C09060=1109.197,421.737,-96.001,-178.441,16.180,151.104
C09061=1109.203,421.984,-96.041,-178.440,16.187,151.106
C09062=1109.209,422.230,-96.081,-178.439,16.194,151.107
C09063=1109.215,422.477,-96.120,-178.437,16.202,151.109
C09064=1109.220,422.724,-96.160,-178.435,16.209,151.110
C09065=1109.225,422.971,-96.199,-178.434,16.216,151.112
C09066=1109.231,423.218,-96.238,-178.433,16.223,151.113
C09067=1109.237,423.436,-96.273,-178.432,16.230,151.115
C09068=1109.241,423.654,-96.308,-178.430,16.237,151.116
C09069=1109.246,423.872,-96.343,-178.429,16.244,151.118
C09070=1109.251,424.090,-96.378,-178.428,16.250,151.119
C09071=1109.256,424.309,-96.413,-178.426,16.257,151.120
C09072=1109.261,424.526,-96.448,-178.425,16.264,151.122
C09073=1109.266,424.744,-96.483,-178.424,16.270,151.123
C09074=1109.271,424.962,-96.518,-178.422,16.277,151.125
C09075=1109.276,425.209,-96.558,-178.421,16.285,151.127
C09076=1109.282,425.456,-96.597,-178.420,16.292,151.128
C09077=1109.287,425.703,-96.637,-178.419,16.300,151.130
C09078=1109.293,425.949,-96.677,-178.418,16.308,151.132
C09079=1109.299,426.196,-96.716,-178.416,16.316,151.133
C09080=1109.304,426.443,-96.756,-178.415,16.323,151.135
C09081=1109.310,426.689,-96.796,-178.413,16.331,151.137
C09082=1109.315,426.936,-96.836,-178.412,16.339,151.139
C09083=1109.320,427.183,-96.875,-178.411,16.347,151.140
C09084=1109.327,427.429,-96.915,-178.409,16.355,151.142
C09085=1109.332,427.676,-96.955,-178.408,16.363,151.144
C09086=1109.338,427.923,-96.995,-178.407,16.371,151.146
C09087=1109.343,428.169,-97.035,-178.406,16.379,151.147
C09088=1109.349,428.416,-97.075,-178.404,16.387,151.149
C09089=1109.354,428.663,-97.115,-178.403,16.395,151.151
C09090=1109.360,428.909,-97.155,-178.402,16.403,151.153
C09091=1109.366,429.157,-97.195,-178.401,16.411,151.155
C09092=1109.371,429.402,-97.235,-178.400,16.419,151.156
C09093=1109.377,429.650,-97.275,-178.398,16.427,151.158
C09094=1109.383,429.896,-97.315,-178.397,16.436,151.160
C09095=1109.388,430.142,-97.355,-178.396,16.444,151.162
C09096=1109.394,430.390,-97.395,-178.395,16.452,151.164
C09097=1109.399,430.636,-97.435,-178.394,16.460,151.166
C09098=1109.405,430.883,-97.475,-178.393,16.469,151.168
C09099=1109.410,431.129,-97.515,-178.392,16.477,151.170
C09100=1109.416,431.376,-97.555,-178.391,16.485,151.172
C09101=1109.422,431.623,-97.596,-178.389,16.495,151.174
C09102=1109.427,431.869,-97.635,-178.388,16.503,151.176
C09103=1109.433,432.116,-97.676,-178.387,16.511,151.178
C09104=1109.438,432.362,-97.716,-178.387,16.520,151.180
C09105=1109.444,432.609,-97.756,-178.386,16.528,151.182
C09106=1109.449,432.856,-97.797,-178.385,16.537,151.184
C09107=1109.455,433.102,-97.837,-178.384,16.545,151.186
C09108=1109.461,433.349,-97.877,-178.383,16.554,151.188
C09109=1109.467,433.595,-97.918,-178.381,16.563,151.190
C09110=1109.472,433.842,-97.958,-178.381,16.572,151.192
C09111=1109.477,434.089,-97.998,-178.380,16.580,151.194
C09112=1109.483,434.335,-98.038,-178.379,16.589,151.196
C09113=1109.488,434.582,-98.079,-178.378,16.597,151.198
C09114=1109.494,434.828,-98.119,-178.377,16.607,151.200
C09115=1109.499,435.075,-98.160,-178.376,16.616,151.202
C09116=1109.505,435.321,-98.201,-178.375,16.624,151.204
C09117=1109.510,435.568,-98.241,-178.375,16.633,151.206
C09118=1109.516,435.814,-98.281,-178.374,16.643,151.208
C09119=1109.522,436.061,-98.322,-178.373,16.652,151.211
C09120=1109.527,436.307,-98.362,-178.372,16.661,151.213
C09121=1109.532,436.554,-98.403,-178.371,16.670,151.215
C09122=1109.538,436.801,-98.444,-178.370,16.679,151.217
C09123=1109.544,437.031,-98.481,-178.369,16.688,151.219
C09124=1109.548,437.262,-98.519,-178.369,16.696,151.221
C09125=1109.553,437.492,-98.558,-178.369,16.704,151.223
C09126=1109.559,437.722,-98.596,-178.368,16.713,151.225
C09127=1109.564,437.953,-98.634,-178.367,16.722,151.227
C09128=1109.570,438.184,-98.672,-178.366,16.731,151.230
C09129=1109.574,438.414,-98.710,-178.366,16.739,151.232
C09130=1109.580,438.646,-98.748,-178.365,16.748,151.234
C09131=1109.585,438.892,-98.789,-178.365,16.758,151.236
C09132=1109.591,439.138,-98.830,-178.363,16.767,151.238
C09133=1109.597,439.385,-98.870,-178.363,16.776,151.241
C09134=1109.602,439.631,-98.911,-178.362,16.786,151.243
C09135=1109.608,439.878,-98.952,-178.362,16.796,151.246
C09136=1109.614,440.124,-98.993,-178.362,16.805,151.248
C09137=1109.619,440.371,-99.034,-178.360,16.815,151.250
C09138=1109.625,440.617,-99.074,-178.360,16.824,151.252
C09139=1109.630,440.863,-99.116,-178.359,16.835,151.255
C09140=1109.636,441.110,-99.156,-178.359,16.844,151.257
C09141=1109.641,441.357,-99.198,-178.359,16.853,151.260
C09142=1109.647,441.603,-99.239,-178.358,16.864,151.262
C09143=1109.652,441.849,-99.279,-178.358,16.873,151.265
C09144=1109.658,442.096,-99.320,-178.357,16.884,151.267
C09145=1109.664,442.342,-99.362,-178.357,16.893,151.270
C09146=1109.669,442.589,-99.402,-178.356,16.904,151.272
C09147=1109.675,442.835,-99.443,-178.356,16.913,151.275
C09148=1109.680,443.081,-99.484,-178.355,16.924,151.277
C09149=1109.685,443.328,-99.526,-178.355,16.933,151.280
C09150=1109.691,443.575,-99.567,-178.355,16.944,151.282
C09151=1109.696,443.820,-99.608,-178.355,16.954,151.285
C09152=1109.702,444.067,-99.649,-178.355,16.964,151.287
C09153=1109.707,444.314,-99.691,-178.355,16.974,151.290
C09154=1109.713,444.560,-99.732,-178.355,16.984,151.293
C09155=1109.719,444.807,-99.773,-178.356,16.994,151.295
C09156=1109.725,445.053,-99.815,-178.356,17.004,151.298
C09157=1109.729,445.299,-99.856,-178.356,17.014,151.301
C09158=1109.735,445.545,-99.897,-178.357,17.024,151.303
C09159=1109.741,445.792,-99.938,-178.358,17.034,151.306
C09160=1109.747,446.038,-99.979,-178.359,17.044,151.309
C09161=1109.752,446.285,-100.021,-178.360,17.053,151.311
C09162=1109.757,446.532,-100.062,-178.361,17.064,151.314
C09163=1109.763,446.778,-100.104,-178.362,17.074,151.317
C09164=1109.768,447.024,-100.145,-178.363,17.084,151.320
C09165=1109.774,447.270,-100.187,-178.364,17.093,151.323
C09166=1109.779,447.517,-100.228,-178.366,17.103,151.326
C09167=1109.785,447.763,-100.269,-178.367,17.113,151.328
C09168=1109.790,448.010,-100.311,-178.369,17.123,151.331
C09169=1109.796,448.257,-100.352,-178.371,17.133,151.334
C09170=1109.802,448.503,-100.394,-178.372,17.143,151.337
C09171=1109.807,448.749,-100.436,-178.375,17.152,151.340
C09172=1109.813,448.996,-100.477,-178.377,17.162,151.343
C09173=1109.817,449.242,-100.518,-178.378,17.172,151.346
C09174=1109.823,449.488,-100.560,-178.381,17.182,151.349
C09175=1109.828,449.735,-100.602,-178.383,17.191,151.352
C09176=1109.834,449.981,-100.643,-178.384,17.201,151.355
C09177=1109.839,450.228,-100.684,-178.387,17.211,151.358
C09178=1109.845,450.474,-100.726,-178.389,17.221,151.361
C09179=1109.435,450.467,-100.832,-178.476,17.454,151.438
C09180=1109.430,450.221,-100.790,-178.473,17.444,151.435
C09181=1109.424,449.975,-100.749,-178.471,17.435,151.432
C09182=1109.419,449.729,-100.707,-178.469,17.424,151.429
C09183=1109.413,449.483,-100.665,-178.467,17.414,151.426
C09184=1109.408,449.235,-100.624,-178.465,17.405,151.423
C09185=1109.402,448.989,-100.582,-178.463,17.395,151.420
C09186=1109.397,448.743,-100.540,-178.461,17.385,151.417
C09187=1109.391,448.496,-100.499,-178.459,17.375,151.414
C09188=1109.386,448.250,-100.457,-178.458,17.365,151.411
C09189=1109.380,448.003,-100.416,-178.456,17.355,151.409
C09190=1109.374,447.757,-100.375,-178.454,17.345,151.406
C09191=1109.369,447.510,-100.333,-178.453,17.335,151.403
C09192=1109.363,447.264,-100.291,-178.451,17.325,151.400
C09193=1109.358,447.017,-100.250,-178.450,17.316,151.397
C09194=1109.353,446.772,-100.209,-178.449,17.306,151.394
C09195=1109.348,446.525,-100.167,-178.448,17.295,151.391
C09196=1109.342,446.279,-100.125,-178.447,17.285,151.389
C09197=1109.336,446.032,-100.084,-178.446,17.275,151.386
C09198=1109.331,445.785,-100.042,-178.445,17.265,151.383
C09199=1109.325,445.539,-100.001,-178.444,17.255,151.380
C09200=1109.319,445.292,-99.960,-178.443,17.245,151.378
C09201=1109.314,445.046,-99.918,-178.443,17.235,151.375
C09202=1109.308,444.800,-99.877,-178.443,17.225,151.372
C09203=1109.303,444.554,-99.836,-178.443,17.215,151.370
C09204=1109.297,444.307,-99.795,-178.443,17.205,151.367
C09205=1109.292,444.061,-99.753,-178.442,17.195,151.364
C09206=1109.286,443.814,-99.712,-178.442,17.184,151.362
C09207=1109.280,443.568,-99.671,-178.442,17.174,151.359
C09208=1109.275,443.321,-99.630,-178.443,17.164,151.357
C09209=1109.270,443.075,-99.588,-178.443,17.154,151.354
C09210=1109.264,442.828,-99.547,-178.444,17.143,151.352
C09211=1109.258,442.582,-99.506,-178.444,17.134,151.349
C09212=1109.253,442.336,-99.464,-178.445,17.124,151.347
C09213=1109.247,442.089,-99.424,-178.445,17.114,151.344
C09214=1109.242,441.844,-99.383,-178.446,17.103,151.342
C09215=1109.236,441.597,-99.342,-178.446,17.094,151.339
C09216=1109.231,441.350,-99.301,-178.447,17.083,151.337
C09217=1109.225,441.104,-99.259,-178.447,17.074,151.334
C09218=1109.220,440.857,-99.219,-178.448,17.064,151.332
C09219=1109.214,440.611,-99.177,-178.448,17.054,151.329
C09220=1109.208,440.364,-99.137,-178.449,17.044,151.327
C09221=1109.203,440.118,-99.096,-178.449,17.034,151.325
C09222=1109.197,439.871,-99.054,-178.451,17.025,151.322
C09223=1109.192,439.625,-99.014,-178.451,17.015,151.320
C09224=1109.186,439.378,-98.973,-178.451,17.006,151.318
C09225=1109.180,439.132,-98.932,-178.452,16.996,151.315
C09226=1109.175,438.885,-98.891,-178.453,16.987,151.313
C09227=1109.169,438.639,-98.851,-178.454,16.977,151.311
C09228=1109.164,438.410,-98.812,-178.454,16.968,151.309
C09229=1109.159,438.181,-98.774,-178.455,16.960,151.306
C09230=1109.153,437.952,-98.737,-178.455,16.951,151.304
C09231=1109.148,437.721,-98.699,-178.456,16.942,151.302
C09232=1109.143,437.492,-98.661,-178.457,16.933,151.300
C09233=1109.138,437.263,-98.623,-178.458,16.924,151.298
C09234=1109.133,437.034,-98.585,-178.458,16.916,151.296
C09235=1109.128,436.805,-98.547,-178.459,16.907,151.294
C09236=1109.122,436.558,-98.506,-178.460,16.898,151.292
C09237=1109.116,436.311,-98.465,-178.461,16.889,151.289
C09238=1109.110,436.065,-98.425,-178.462,16.879,151.287
C09239=1109.105,435.819,-98.385,-178.463,16.871,151.285
C09240=1109.099,435.572,-98.344,-178.463,16.862,151.283
C09241=1109.094,435.325,-98.303,-178.465,16.852,151.281
C09242=1109.089,435.079,-98.263,-178.466,16.843,151.279
C09243=1109.083,434.832,-98.222,-178.466,16.834,151.277
C09244=1109.077,434.585,-98.182,-178.467,16.825,151.274
C09245=1109.072,434.339,-98.141,-178.468,16.816,151.272
C09246=1109.066,434.092,-98.101,-178.469,16.807,151.270
C09247=1109.061,433.846,-98.061,-178.470,16.799,151.268
C09248=1109.056,433.599,-98.021,-178.471,16.790,151.266
C09249=1109.050,433.352,-97.980,-178.472,16.780,151.264
C09250=1109.044,433.106,-97.940,-178.473,16.772,151.262
C09251=1109.039,432.859,-97.899,-178.474,16.763,151.260
C09252=1109.033,432.613,-97.859,-178.475,16.755,151.258
C09253=1109.028,432.367,-97.818,-178.476,16.746,151.256
C09254=1109.022,432.120,-97.778,-178.477,16.738,151.254
C09255=1109.016,431.873,-97.738,-178.479,16.729,151.252
C09256=1109.011,431.626,-97.698,-178.480,16.720,151.250
C09257=1109.005,431.380,-97.658,-178.481,16.712,151.248
C09258=1109.000,431.134,-97.617,-178.482,16.703,151.246
C09259=1108.994,430.887,-97.578,-178.483,16.695,151.244
C09260=1108.988,430.640,-97.537,-178.484,16.687,151.242
C09261=1108.983,430.394,-97.497,-178.485,16.678,151.240
C09262=1108.977,430.147,-97.457,-178.486,16.670,151.239
C09263=1108.972,429.900,-97.417,-178.487,16.662,151.237
C09264=1108.966,429.654,-97.376,-178.489,16.653,151.235
C09265=1108.960,429.406,-97.337,-178.490,16.645,151.233
C09266=1108.955,429.160,-97.296,-178.491,16.636,151.231
C09267=1108.949,428.913,-97.257,-178.493,16.628,151.229
C09268=1108.944,428.667,-97.216,-178.494,16.620,151.227
C09269=1108.938,428.420,-97.177,-178.495,16.612,151.225
C09270=1108.932,428.173,-97.136,-178.496,16.604,151.224
C09271=1108.926,427.927,-97.097,-178.497,16.596,151.222
C09272=1108.921,427.680,-97.057,-178.499,16.588,151.220
C09273=1108.916,427.433,-97.017,-178.500,16.580,151.218
C09274=1108.909,427.187,-96.977,-178.501,16.572,151.216
C09275=1108.905,426.940,-96.938,-178.503,16.564,151.215
C09276=1108.898,426.694,-96.897,-178.504,16.556,151.213
C09277=1108.893,426.446,-96.857,-178.505,16.548,151.211
C09278=1108.887,426.200,-96.818,-178.507,16.540,151.210
C09279=1108.882,425.953,-96.778,-178.508,16.532,151.208
C09280=1108.876,425.707,-96.739,-178.509,16.525,151.206
C09281=1108.870,425.460,-96.698,-178.510,16.517,151.204
C09282=1108.865,425.213,-96.659,-178.512,16.509,151.203
C09283=1108.859,424.966,-96.619,-178.513,16.501,151.201
C09284=1108.854,424.748,-96.584,-178.514,16.495,151.199
C09285=1108.849,424.530,-96.549,-178.516,16.487,151.198
C09286=1108.845,424.312,-96.514,-178.517,16.481,151.197
C09287=1108.840,424.094,-96.479,-178.518,16.474,151.195
C09288=1108.835,423.876,-96.444,-178.519,16.467,151.194
C09289=1108.830,423.657,-96.409,-178.521,16.460,151.192
C09290=1108.825,423.439,-96.374,-178.522,16.454,151.191
C09291=1108.820,423.222,-96.339,-178.524,16.447,151.189
C09292=1108.814,422.974,-96.299,-178.525,16.439,151.188
C09293=1108.809,422.728,-96.260,-178.527,16.432,151.186
C09294=1108.803,422.480,-96.220,-178.528,16.425,151.184
C09295=1108.798,422.234,-96.181,-178.529,16.417,151.183
C09296=1108.792,421.987,-96.142,-178.531,16.410,151.181
C09297=1108.786,421.740,-96.103,-178.533,16.403,151.180
C09298=1108.780,421.493,-96.063,-178.535,16.395,151.178
C09299=1108.775,421.247,-96.024,-178.535,16.388,151.177
C09300=1108.769,421.000,-95.983,-178.537,16.381,151.175
C09301=1108.764,420.754,-95.944,-178.539,16.373,151.174
C09302=1108.757,420.507,-95.905,-178.541,16.366,151.172
C09303=1108.752,420.260,-95.866,-178.542,16.359,151.171
C09304=1108.746,420.012,-95.827,-178.544,16.352,151.169
C09305=1108.742,419.766,-95.787,-178.545,16.345,151.168
C09306=1108.736,419.519,-95.748,-178.547,16.337,151.166
C09307=1108.730,419.272,-95.709,-178.548,16.331,151.165
C09308=1108.724,419.026,-95.670,-178.550,16.323,151.163
C09309=1108.718,418.778,-95.630,-178.552,16.316,151.162
C09310=1108.713,418.532,-95.591,-178.553,16.309,151.160
C09311=1108.707,418.286,-95.552,-178.555,16.302,151.159
C09312=1108.701,418.038,-95.513,-178.557,16.295,151.157
C09313=1108.696,417.791,-95.475,-178.558,16.289,151.156
C09314=1108.691,417.544,-95.435,-178.560,16.281,151.155
C09315=1108.685,417.298,-95.395,-178.562,16.274,151.153
C09316=1108.680,417.051,-95.356,-178.563,16.268,151.152
C09317=1108.674,416.803,-95.318,-178.565,16.261,151.150
C09318=1108.669,416.557,-95.279,-178.566,16.254,151.149
C09319=1108.663,416.310,-95.239,-178.568,16.247,151.148
C09320=1108.657,416.063,-95.200,-178.570,16.240,151.146
C09321=1108.651,415.817,-95.162,-178.572,16.234,151.145
C09322=1108.645,415.569,-95.123,-178.574,16.227,151.144
C09323=1108.640,415.323,-95.084,-178.575,16.221,151.142
C09324=1108.634,415.075,-95.045,-178.577,16.213,151.141
C09325=1108.628,414.829,-95.006,-178.578,16.207,151.139
C09326=1108.623,414.582,-94.968,-178.581,16.200,151.138
C09327=1108.617,414.335,-94.928,-178.583,16.193,151.137
C09328=1108.612,414.088,-94.889,-178.584,16.187,151.136
C09329=1108.606,413.841,-94.851,-178.586,16.180,151.134
C09330=1108.600,413.594,-94.812,-178.588,16.174,151.133
C09331=1108.595,413.347,-94.774,-178.590,16.168,151.132
C09332=1108.589,413.101,-94.735,-178.591,16.161,151.131
C09333=1108.583,412.853,-94.696,-178.593,16.155,151.129
C09334=1108.578,412.607,-94.657,-178.595,16.148,151.128
C09335=1108.572,412.360,-94.619,-178.597,16.142,151.127
C09336=1108.566,412.113,-94.580,-178.599,16.135,151.125
C09337=1108.561,411.866,-94.541,-178.600,16.129,151.124
C09338=1108.556,411.619,-94.503,-178.603,16.123,151.123
C09339=1108.550,411.372,-94.464,-178.604,16.117,151.122
C09340=1108.545,411.160,-94.431,-178.606,16.111,151.121
C09341=1108.540,410.948,-94.398,-178.607,16.106,151.120
C09342=1108.535,410.736,-94.364,-178.609,16.100,151.119
C09343=1108.531,410.525,-94.332,-178.611,16.095,151.118
C09344=1108.526,410.313,-94.299,-178.612,16.090,151.117
C09345=1108.521,410.101,-94.266,-178.614,16.084,151.116
C09346=1108.516,409.890,-94.233,-178.616,16.079,151.115
C09347=1108.511,409.678,-94.200,-178.617,16.074,151.114
C09348=1108.506,409.431,-94.161,-178.620,16.067,151.113
C09349=1108.501,409.184,-94.123,-178.621,16.061,151.111
C09350=1108.495,408.936,-94.084,-178.623,16.055,151.110
C09351=1108.489,408.690,-94.046,-178.625,16.049,151.109
C09352=1108.483,408.443,-94.008,-178.627,16.043,151.108
C09353=1108.478,408.196,-93.969,-178.629,16.037,151.107
C09354=1108.472,407.949,-93.931,-178.631,16.031,151.106
C09355=1108.467,407.702,-93.893,-178.633,16.025,151.105
C09356=1108.461,407.455,-93.854,-178.635,16.019,151.104
C09357=1108.455,407.208,-93.816,-178.636,16.014,151.103
C09358=1108.450,406.961,-93.778,-178.639,16.007,151.101
C09359=1108.444,406.714,-93.739,-178.641,16.001,151.100
C09360=1108.438,406.467,-93.701,-178.642,15.996,151.099
C09361=1108.433,406.220,-93.663,-178.644,15.990,151.098
C09362=1108.427,405.973,-93.625,-178.647,15.984,151.097
C09363=1108.422,405.726,-93.587,-178.649,15.978,151.096
C09364=1108.416,405.479,-93.549,-178.650,15.972,151.095
C09365=1108.411,405.232,-93.510,-178.652,15.967,151.094
C09366=1108.405,404.985,-93.472,-178.655,15.961,151.093
C09367=1108.399,404.738,-93.434,-178.657,15.955,151.092
C09368=1108.394,404.491,-93.396,-178.659,15.949,151.091
C09369=1108.388,404.244,-93.359,-178.661,15.944,151.090
C09370=1108.382,403.997,-93.320,-178.663,15.938,151.089
C09371=1108.376,403.750,-93.282,-178.665,15.933,151.088
C09372=1108.371,403.503,-93.244,-178.667,15.927,151.087
C09373=1108.365,403.256,-93.206,-178.669,15.921,151.086
C09374=1108.360,403.008,-93.168,-178.671,15.916,151.085
C09375=1108.354,402.762,-93.131,-178.673,15.910,151.084
C09376=1108.348,402.515,-93.093,-178.675,15.905,151.083
C09377=1108.343,402.268,-93.054,-178.677,15.899,151.082
C09378=1108.337,402.021,-93.017,-178.679,15.894,151.081
C09379=1108.331,401.773,-92.979,-178.681,15.888,151.080
C09380=1108.326,401.526,-92.941,-178.683,15.883,151.080
C09381=1108.320,401.279,-92.903,-178.686,15.877,151.078
C09382=1108.314,401.032,-92.865,-178.688,15.871,151.078
C09383=1108.309,400.785,-92.828,-178.690,15.866,151.077
C09384=1108.303,400.538,-92.790,-178.692,15.861,151.076
C09385=1108.297,400.291,-92.752,-178.695,15.856,151.075
C09386=1108.292,400.044,-92.714,-178.697,15.850,151.074
C09387=1108.287,399.797,-92.677,-178.699,15.845,151.073
C09388=1108.281,399.550,-92.639,-178.701,15.840,151.072
C09389=1108.275,399.303,-92.601,-178.703,15.834,151.071
C09390=1108.270,399.056,-92.564,-178.705,15.829,151.070
C09391=1108.264,398.809,-92.526,-178.707,15.824,151.070
C09392=1108.258,398.561,-92.489,-178.710,15.819,151.069
C09393=1108.252,398.315,-92.451,-178.712,15.814,151.068
C09394=1108.247,398.068,-92.413,-178.714,15.808,151.067
C09395=1108.242,397.820,-92.376,-178.716,15.803,151.066
C09396=1108.236,397.609,-92.343,-178.718,15.799,151.066
C09397=1108.232,397.396,-92.311,-178.720,15.795,151.065
C09398=1108.227,397.185,-92.279,-178.722,15.790,151.064
C09399=1108.222,396.972,-92.247,-178.724,15.786,151.063
C09400=1108.217,396.760,-92.216,-178.726,15.781,151.063
C09401=1108.212,396.548,-92.183,-178.727,15.777,151.062
C09402=1108.208,396.336,-92.151,-178.730,15.772,151.061
C09403=1108.203,396.124,-92.118,-178.732,15.768,151.061
C09404=1108.197,395.877,-92.081,-178.734,15.763,151.060
C09405=1108.191,395.630,-92.043,-178.736,15.758,151.059
C09406=1108.186,395.383,-92.006,-178.739,15.753,151.058
C09407=1108.180,395.135,-91.969,-178.741,15.748,151.058
C09408=1108.174,394.889,-91.932,-178.742,15.744,151.057
C09409=1108.169,394.641,-91.895,-178.745,15.739,151.056
C09410=1108.163,394.395,-91.857,-178.747,15.734,151.055
C09411=1108.158,394.148,-91.820,-178.750,15.729,151.055
C09412=1108.152,393.901,-91.783,-178.752,15.724,151.054
C09413=1108.146,393.654,-91.745,-178.754,15.719,151.053
C09414=1108.141,393.406,-91.708,-178.757,15.714,151.053
C09415=1108.135,393.159,-91.671,-178.759,15.709,151.052
C09416=1108.129,392.912,-91.634,-178.762,15.704,151.051
C09417=1108.123,392.665,-91.596,-178.763,15.700,151.050
C09418=1108.118,392.418,-91.559,-178.766,15.695,151.050
C09419=1108.112,392.170,-91.522,-178.768,15.691,151.049
C09420=1108.106,391.923,-91.486,-178.771,15.686,151.048
C09421=1108.101,391.677,-91.449,-178.773,15.681,151.048
C09422=1108.095,391.430,-91.412,-178.776,15.676,151.047
C09423=1108.089,391.182,-91.374,-178.778,15.672,151.046
C09424=1108.084,390.935,-91.337,-178.780,15.667,151.046
C09425=1108.078,390.688,-91.300,-178.783,15.662,151.045
C09426=1108.072,390.441,-91.264,-178.785,15.657,151.044
C09427=1108.066,390.194,-91.226,-178.788,15.653,151.044
C09428=1108.061,389.947,-91.190,-178.790,15.649,151.043
C09429=1108.055,389.700,-91.152,-178.792,15.644,151.042
C09430=1108.050,389.452,-91.115,-178.795,15.639,151.042
C09431=1108.043,389.205,-91.079,-178.797,15.635,151.041
C09432=1108.038,388.958,-91.042,-178.800,15.630,151.041
C09433=1108.033,388.711,-91.005,-178.802,15.626,151.040
C09434=1108.027,388.464,-90.969,-178.805,15.621,151.039
C09435=1108.021,388.217,-90.932,-178.807,15.617,151.039
C09436=1108.015,387.970,-90.895,-178.810,15.612,151.038
C09437=1108.010,387.722,-90.858,-178.812,15.608,151.038
C09438=1108.004,387.476,-90.822,-178.815,15.604,151.037
C09439=1107.998,387.229,-90.785,-178.817,15.599,151.037
C09440=1107.993,386.981,-90.748,-178.820,15.594,151.036
C09441=1107.986,386.734,-90.711,-178.822,15.590,151.035
C09442=1107.981,386.487,-90.674,-178.825,15.586,151.035
C09443=1107.976,386.240,-90.637,-178.827,15.581,151.034
C09444=1107.971,385.992,-90.601,-178.830,15.577,151.034
C09445=1107.965,385.746,-90.565,-178.832,15.573,151.033
C09446=1107.959,385.498,-90.528,-178.835,15.568,151.033
C09447=1107.953,385.251,-90.492,-178.838,15.564,151.032
C09448=1107.947,385.004,-90.454,-178.840,15.559,151.032
C09449=1107.943,384.757,-90.419,-178.842,15.555,151.031
C09450=1107.936,384.510,-90.382,-178.845,15.551,151.030
C09451=1107.931,384.262,-90.345,-178.848,15.546,151.030
C09452=1107.921,383.851,-90.284,-178.852,15.540,151.029
C09453=1107.912,383.439,-90.223,-178.856,15.533,151.028
C09454=1107.903,383.027,-90.162,-178.861,15.526,151.027
C09455=1107.893,382.615,-90.103,-178.865,15.519,151.027
C09456=1107.888,382.367,-90.065,-178.867,15.515,151.026
C09457=1107.882,382.121,-90.029,-178.870,15.511,151.026
C09458=1107.877,381.873,-89.993,-178.873,15.506,151.025
C09459=1107.871,381.626,-89.957,-178.875,15.502,151.025
C09460=1107.865,381.379,-89.921,-178.878,15.498,151.024
C09461=1107.859,381.131,-89.884,-178.881,15.494,151.024
C09462=1107.853,380.884,-89.848,-178.883,15.490,151.023
C09463=1107.848,380.637,-89.812,-178.886,15.486,151.023
C09464=1107.842,380.390,-89.775,-178.888,15.483,151.023
C09465=1107.836,380.142,-89.740,-178.891,15.478,151.022
C09466=1107.831,379.896,-89.703,-178.894,15.474,151.022
C09467=1107.825,379.648,-89.667,-178.896,15.470,151.021
C09468=1107.819,379.401,-89.630,-178.899,15.466,151.021
C09469=1107.814,379.154,-89.595,-178.902,15.463,151.021
C09470=1107.808,378.906,-89.559,-178.905,15.458,151.020
C09471=1107.803,378.659,-89.522,-178.907,15.455,151.020
C09472=1107.797,378.412,-89.487,-178.910,15.451,151.019
C09473=1107.791,378.165,-89.450,-178.913,15.446,151.019
C09474=1107.786,377.917,-89.414,-178.915,15.443,151.019
C09475=1107.780,377.670,-89.379,-178.918,15.439,151.018
C09476=1107.774,377.423,-89.343,-178.921,15.435,151.018
C09477=1107.769,377.175,-89.306,-178.924,15.431,151.017
C09478=1107.763,376.928,-89.271,-178.926,15.428,151.017
C09479=1107.757,376.681,-89.234,-178.929,15.423,151.017
C09480=1107.752,376.433,-89.198,-178.931,15.420,151.016
C09481=1107.746,376.186,-89.163,-178.934,15.416,151.016
C09482=1107.740,375.939,-89.127,-178.937,15.413,151.016
C09483=1107.735,375.692,-89.091,-178.940,15.408,151.015
C09484=1107.729,375.444,-89.055,-178.942,15.405,151.015
C09485=1107.724,375.197,-89.019,-178.945,15.401,151.014
C09486=1107.718,374.950,-88.983,-178.948,15.398,151.014
C09487=1107.712,374.703,-88.948,-178.951,15.393,151.014
C09488=1107.707,374.455,-88.911,-178.953,15.390,151.014
C09489=1107.701,374.208,-88.876,-178.956,15.386,151.013
C09490=1107.695,373.961,-88.840,-178.959,15.383,151.013
C09491=1107.690,373.714,-88.805,-178.962,15.379,151.013
C09492=1107.684,373.466,-88.769,-178.964,15.375,151.012
C09493=1107.679,373.219,-88.734,-178.968,15.371,151.012
C09494=1107.672,372.971,-88.698,-178.970,15.368,151.012
C09495=1107.667,372.724,-88.662,-178.973,15.364,151.011
C09496=1107.661,372.477,-88.627,-178.976,15.361,151.011
C09497=1107.656,372.229,-88.590,-178.979,15.357,151.011
C09498=1107.650,371.982,-88.555,-178.982,15.354,151.011
C09499=1107.644,371.734,-88.519,-178.984,15.350,151.010
C09500=1107.639,371.487,-88.484,-178.987,15.347,151.010
C09501=1107.633,371.239,-88.448,-178.990,15.344,151.010
C09502=1107.627,370.993,-88.413,-178.993,15.339,151.010
C09503=1107.622,370.746,-88.377,-178.996,15.336,151.009
C09504=1107.613,370.360,-88.322,-179.000,15.331,151.009
C09505=1107.604,369.975,-88.267,-179.005,15.325,151.009
C09506=1107.595,369.590,-88.211,-179.009,15.320,151.008
C09507=1107.586,369.204,-88.156,-179.014,15.314,151.008
C09508=1107.581,368.957,-88.121,-179.016,15.311,151.008
C09509=1107.575,368.710,-88.085,-179.019,15.308,151.007
C09510=1107.570,368.462,-88.050,-179.022,15.304,151.007
C09511=1107.564,368.215,-88.015,-179.025,15.301,151.007
C09512=1107.558,367.967,-87.979,-179.028,15.298,151.007
C09513=1107.553,367.720,-87.944,-179.031,15.294,151.007
C09514=1107.548,367.472,-87.909,-179.034,15.291,151.006
C09515=1107.541,367.225,-87.874,-179.037,15.287,151.006
C09516=1107.535,366.978,-87.839,-179.040,15.284,151.006
C09517=1107.529,366.730,-87.803,-179.042,15.281,151.006
C09518=1107.524,366.483,-87.768,-179.046,15.278,151.006
C09519=1107.519,366.236,-87.733,-179.048,15.274,151.005
C09520=1107.513,365.988,-87.697,-179.051,15.271,151.005
C09521=1107.508,365.741,-87.663,-179.055,15.268,151.005
C09522=1107.502,365.494,-87.627,-179.057,15.265,151.005
C09523=1107.496,365.246,-87.593,-179.060,15.262,151.005
C09524=1107.490,364.999,-87.557,-179.063,15.258,151.005
C09525=1107.484,364.751,-87.522,-179.066,15.255,151.004
C09526=1107.479,364.503,-87.487,-179.069,15.252,151.004
C09527=1107.474,364.256,-87.452,-179.072,15.248,151.004
C09528=1107.467,364.008,-87.417,-179.075,15.246,151.004
C09529=1107.462,363.761,-87.382,-179.078,15.243,151.004
C09530=1107.457,363.514,-87.347,-179.081,15.240,151.004
C09531=1107.451,363.266,-87.312,-179.084,15.236,151.004
C09532=1107.445,363.019,-87.277,-179.087,15.233,151.004
C09533=1107.439,362.772,-87.242,-179.090,15.230,151.003
C09534=1107.434,362.524,-87.207,-179.093,15.227,151.003
C09535=1107.427,362.277,-87.172,-179.096,15.224,151.003
C09536=1107.422,362.029,-87.138,-179.099,15.221,151.003
C09537=1107.417,361.781,-87.103,-179.102,15.218,151.003
C09538=1107.410,361.534,-87.068,-179.105,15.214,151.003
C09539=1107.405,361.287,-87.033,-179.108,15.211,151.003
C09540=1107.400,361.038,-86.998,-179.111,15.209,151.003
C09541=1107.393,360.792,-86.963,-179.114,15.205,151.003
C09542=1107.388,360.544,-86.929,-179.117,15.202,151.002
C09543=1107.383,360.297,-86.894,-179.120,15.199,151.002
C09544=1107.376,360.049,-86.859,-179.123,15.197,151.002
C09545=1107.371,359.802,-86.824,-179.127,15.193,151.002
C09546=1107.365,359.554,-86.790,-179.129,15.190,151.002
C09547=1107.360,359.306,-86.755,-179.132,15.188,151.002
C09548=1107.354,359.059,-86.720,-179.135,15.185,151.002
C09549=1107.348,358.812,-86.686,-179.138,15.182,151.002
C09550=1107.343,358.564,-86.651,-179.142,15.179,151.002
C09551=1107.337,358.316,-86.617,-179.145,15.176,151.002
C09552=1107.332,358.069,-86.582,-179.148,15.173,151.002
C09553=1107.326,357.822,-86.547,-179.151,15.171,151.002
C09554=1107.320,357.574,-86.512,-179.153,15.168,151.002
C09555=1107.314,357.326,-86.478,-179.157,15.164,151.002
C09556=1107.306,356.955,-86.426,-179.162,15.160,151.002
C09557=1107.297,356.586,-86.375,-179.166,15.156,151.002
C09558=1107.288,356.215,-86.324,-179.171,15.151,151.002
C09559=1107.280,355.844,-86.272,-179.175,15.147,151.002
C09560=1107.274,355.597,-86.238,-179.179,15.145,151.002
C09561=1107.269,355.349,-86.203,-179.182,15.142,151.002
C09562=1107.263,355.102,-86.169,-179.184,15.139,151.002
C09563=1107.258,354.854,-86.134,-179.187,15.137,151.002
C09564=1107.252,354.606,-86.100,-179.191,15.133,151.002
C09565=1107.246,354.359,-86.066,-179.194,15.131,151.002
C09566=1107.241,354.111,-86.031,-179.197,15.128,151.002
C09567=1107.235,353.864,-85.997,-179.200,15.125,151.002
C09568=1107.230,353.617,-85.963,-179.203,15.123,151.002
C09569=1107.224,353.369,-85.929,-179.206,15.120,151.002
C09570=1107.218,353.121,-85.895,-179.210,15.117,151.002
C09571=1107.213,352.873,-85.860,-179.213,15.114,151.002
C09572=1107.207,352.626,-85.826,-179.216,15.112,151.002
C09573=1107.201,352.379,-85.792,-179.219,15.109,151.002
C09574=1107.196,352.131,-85.757,-179.222,15.107,151.002
C09575=1107.190,351.883,-85.724,-179.225,15.104,151.002
C09576=1107.184,351.635,-85.690,-179.228,15.101,151.002
C09577=1107.178,351.388,-85.656,-179.232,15.099,151.002
C09578=1107.173,351.140,-85.621,-179.235,15.096,151.002
C09579=1107.167,350.893,-85.587,-179.238,15.093,151.002
C09580=1107.161,350.645,-85.554,-179.242,15.091,151.002
C09581=1107.156,350.398,-85.520,-179.245,15.088,151.002
C09582=1107.150,350.150,-85.485,-179.248,15.086,151.002
C09583=1107.145,349.902,-85.452,-179.251,15.083,151.002
C09584=1107.138,349.654,-85.417,-179.254,15.081,151.002
C09585=1107.133,349.407,-85.383,-179.257,15.078,151.003
C09586=1107.127,349.159,-85.350,-179.260,15.076,151.003
C09587=1107.122,348.911,-85.315,-179.263,15.073,151.003
C09588=1107.116,348.664,-85.281,-179.267,15.071,151.003
C09589=1107.110,348.416,-85.248,-179.270,15.069,151.003
C09590=1107.105,348.169,-85.214,-179.274,15.065,151.003
C09591=1107.099,347.921,-85.180,-179.277,15.063,151.003
C09592=1107.093,347.674,-85.146,-179.280,15.060,151.003
C09593=1107.088,347.426,-85.113,-179.283,15.058,151.003
C09594=1107.083,347.178,-85.078,-179.287,15.056,151.003
C09595=1107.077,346.930,-85.045,-179.290,15.053,151.004
C09596=1107.071,346.683,-85.011,-179.293,15.051,151.004
C09597=1107.066,346.435,-84.978,-179.296,15.048,151.004
C09598=1107.060,346.188,-84.943,-179.299,15.046,151.004
C09599=1107.054,345.940,-84.910,-179.302,15.043,151.004
C09600=1107.048,345.693,-84.876,-179.306,15.041,151.004
C09601=1107.043,345.445,-84.843,-179.309,15.039,151.004
C09602=1107.037,345.198,-84.809,-179.312,15.036,151.004
C09603=1107.031,344.950,-84.775,-179.315,15.034,151.004
C09604=1107.025,344.701,-84.742,-179.319,15.032,151.005
C09605=1107.019,344.454,-84.708,-179.322,15.029,151.005
C09606=1107.014,344.206,-84.674,-179.325,15.027,151.005
C09607=1107.008,343.958,-84.641,-179.328,15.025,151.005
C09608=1107.000,343.590,-84.590,-179.333,15.021,151.005
C09609=1106.991,343.222,-84.541,-179.338,15.018,151.006
C09610=1106.983,342.854,-84.491,-179.343,15.014,151.006
C09611=1106.974,342.485,-84.441,-179.348,15.011,151.006
C09612=1106.969,342.237,-84.408,-179.351,15.008,151.006
C09613=1106.963,341.989,-84.374,-179.355,15.006,151.006
C09614=1106.958,341.741,-84.341,-179.358,15.004,151.007
C09615=1106.951,341.494,-84.308,-179.361,15.002,151.007
C09616=1106.946,341.246,-84.274,-179.365,14.999,151.007
C09617=1106.941,340.999,-84.241,-179.368,14.997,151.007
C09618=1106.935,340.751,-84.208,-179.371,14.995,151.007
C09619=1106.930,340.503,-84.175,-179.375,14.993,151.007
C09620=1106.924,340.255,-84.141,-179.378,14.990,151.007
C09621=1106.918,340.008,-84.107,-179.381,14.989,151.008
C09622=1106.912,339.760,-84.075,-179.384,14.987,151.008
C09623=1106.906,339.513,-84.041,-179.387,14.984,151.008
C09624=1106.901,339.265,-84.008,-179.391,14.982,151.008
C09625=1106.895,339.017,-83.974,-179.394,14.980,151.008
C09626=1106.890,338.769,-83.941,-179.397,14.978,151.009
C09627=1106.883,338.521,-83.908,-179.401,14.976,151.009
C09628=1106.878,338.274,-83.875,-179.404,14.973,151.009
C09629=1106.873,338.026,-83.842,-179.408,14.971,151.009
C09630=1106.867,337.778,-83.809,-179.411,14.969,151.010
C09631=1106.861,337.531,-83.776,-179.415,14.967,151.010
C09632=1106.855,337.283,-83.743,-179.418,14.965,151.010
C09633=1106.850,337.035,-83.709,-179.421,14.963,151.010
C09634=1106.844,336.787,-83.677,-179.424,14.962,151.011
C09635=1106.838,336.539,-83.643,-179.427,14.959,151.011
C09636=1106.833,336.291,-83.611,-179.431,14.957,151.011
C09637=1106.827,336.044,-83.578,-179.434,14.955,151.011
C09638=1106.821,335.796,-83.545,-179.438,14.953,151.011
C09639=1106.816,335.548,-83.512,-179.441,14.951,151.012
C09640=1106.810,335.300,-83.479,-179.445,14.949,151.012
C09641=1106.804,335.053,-83.446,-179.448,14.947,151.012
C09642=1106.799,334.805,-83.412,-179.452,14.945,151.013
C09643=1106.793,334.557,-83.381,-179.454,14.943,151.013
C09644=1106.788,334.309,-83.347,-179.458,14.941,151.013
C09645=1106.781,334.062,-83.314,-179.461,14.939,151.013
C09646=1106.776,333.814,-83.281,-179.465,14.937,151.013
C09647=1106.771,333.565,-83.248,-179.468,14.935,151.014
C09648=1106.765,333.318,-83.216,-179.472,14.933,151.014
C09649=1106.759,333.070,-83.183,-179.475,14.931,151.014
C09650=1106.753,332.822,-83.151,-179.478,14.929,151.014
C09651=1106.748,332.574,-83.117,-179.481,14.927,151.015
C09652=1106.742,332.327,-83.085,-179.485,14.925,151.015
C09653=1106.737,332.079,-83.052,-179.489,14.923,151.015
C09654=1106.730,331.831,-83.020,-179.492,14.921,151.016
C09655=1106.725,331.583,-82.986,-179.496,14.919,151.016
C09656=1106.719,331.335,-82.954,-179.499,14.918,151.016
C09657=1106.713,331.088,-82.922,-179.502,14.916,151.017
C09658=1106.708,330.840,-82.889,-179.506,14.914,151.017
C09659=1106.702,330.592,-82.857,-179.509,14.912,151.017
C09660=1106.693,330.218,-82.807,-179.515,14.909,151.018
C09661=1106.684,329.843,-82.758,-179.519,14.907,151.018
C09662=1106.675,329.469,-82.709,-179.525,14.904,151.019
C09663=1106.667,329.095,-82.660,-179.530,14.901,151.019
C09664=1106.661,328.846,-82.627,-179.534,14.899,151.019
C09665=1106.655,328.598,-82.595,-179.536,14.898,151.020
C09666=1106.649,328.350,-82.562,-179.540,14.896,151.020
C09667=1106.644,328.103,-82.530,-179.544,14.894,151.021
C09668=1106.638,327.855,-82.497,-179.547,14.892,151.021
C09669=1106.632,327.607,-82.465,-179.550,14.891,151.021
C09670=1106.627,327.360,-82.432,-179.554,14.889,151.021
C09671=1106.621,327.111,-82.400,-179.557,14.887,151.022
C09672=1106.615,326.863,-82.368,-179.561,14.885,151.022
C09673=1106.609,326.616,-82.335,-179.565,14.883,151.022
C09674=1106.604,326.368,-82.303,-179.568,14.882,151.023
C09675=1106.598,326.119,-82.271,-179.571,14.880,151.023
C09676=1106.592,325.872,-82.238,-179.575,14.878,151.024
C09677=1106.587,325.624,-82.207,-179.578,14.877,151.024
C09678=1106.581,325.376,-82.174,-179.581,14.875,151.024
C09679=1106.575,325.128,-82.141,-179.585,14.874,151.025
C09680=1106.570,324.881,-82.110,-179.589,14.872,151.025
C09681=1106.564,324.633,-82.078,-179.592,14.870,151.025
C09682=1106.558,324.385,-82.046,-179.595,14.869,151.026
C09683=1106.553,324.136,-82.013,-179.599,14.867,151.026
C09684=1106.547,323.889,-81.981,-179.603,14.865,151.026
C09685=1106.541,323.641,-81.949,-179.606,14.864,151.027
C09686=1106.535,323.393,-81.917,-179.609,14.862,151.027
C09687=1106.530,323.146,-81.885,-179.613,14.860,151.028
C09688=1106.524,322.897,-81.853,-179.617,14.858,151.028
C09689=1106.519,322.649,-81.821,-179.620,14.857,151.028
C09690=1106.513,322.402,-81.788,-179.623,14.855,151.029
C09691=1106.507,322.154,-81.756,-179.627,14.853,151.029
C09692=1106.502,321.906,-81.725,-179.631,14.852,151.029
C09693=1106.496,321.658,-81.693,-179.634,14.851,151.030
C09694=1106.490,321.411,-81.661,-179.637,14.849,151.030
C09695=1106.484,321.162,-81.629,-179.641,14.847,151.031
C09696=1106.479,320.915,-81.597,-179.644,14.846,151.031
C09697=1106.474,320.666,-81.565,-179.648,14.844,151.031
C09698=1106.468,320.419,-81.533,-179.651,14.842,151.032
C09699=1106.462,320.171,-81.501,-179.654,14.841,151.032
C09700=1106.457,319.923,-81.469,-179.658,14.840,151.032
C09701=1106.451,319.675,-81.437,-179.662,14.838,151.033
C09702=1106.446,319.427,-81.406,-179.666,14.836,151.033
C09703=1106.440,319.179,-81.374,-179.669,14.835,151.034
C09704=1106.434,318.932,-81.342,-179.672,14.833,151.034
C09705=1106.428,318.683,-81.310,-179.676,14.831,151.034
C09706=1106.423,318.436,-81.278,-179.679,14.830,151.035
C09707=1106.417,318.187,-81.247,-179.683,14.828,151.035
C09708=1106.412,317.940,-81.215,-179.687,14.827,151.036
C09709=1106.406,317.691,-81.183,-179.690,14.826,151.036
C09710=1106.400,317.444,-81.152,-179.693,14.824,151.037
C09711=1106.394,317.196,-81.120,-179.697,14.822,151.037
C09712=1106.386,316.814,-81.071,-179.702,14.820,151.037
C09713=1106.377,316.433,-81.022,-179.708,14.818,151.038
C09714=1106.370,316.051,-80.973,-179.713,14.815,151.039
C09715=1106.361,315.669,-80.925,-179.718,14.813,151.039
C09716=1106.355,315.422,-80.893,-179.722,14.811,151.040
C09717=1106.349,315.173,-80.862,-179.725,14.811,151.040
C09718=1106.344,314.926,-80.831,-179.729,14.809,151.041
C09719=1106.338,314.678,-80.799,-179.733,14.808,151.041
C09720=1106.333,314.429,-80.768,-179.736,14.807,151.042
C09721=1106.326,314.181,-80.736,-179.740,14.805,151.042
C09722=1106.320,313.934,-80.705,-179.744,14.804,151.043
C09723=1106.315,313.686,-80.674,-179.747,14.802,151.043
C09724=1106.309,313.438,-80.642,-179.751,14.801,151.044
C09725=1106.303,313.190,-80.611,-179.754,14.800,151.044
C09726=1106.298,312.942,-80.579,-179.758,14.798,151.045
C09727=1106.291,312.694,-80.548,-179.762,14.797,151.045
C09728=1106.286,312.446,-80.516,-179.765,14.796,151.045
C09729=1106.280,312.198,-80.485,-179.769,14.794,151.046
C09730=1106.274,311.951,-80.454,-179.772,14.794,151.046
C09731=1106.269,311.702,-80.423,-179.776,14.792,151.047
C09732=1106.263,311.454,-80.391,-179.780,14.790,151.047
C09733=1106.257,311.207,-80.361,-179.783,14.790,151.048
C09734=1106.251,310.958,-80.329,-179.787,14.788,151.048
C09735=1106.246,310.711,-80.298,-179.790,14.787,151.049
C09736=1106.240,310.462,-80.266,-179.794,14.786,151.049
C09737=1106.235,310.214,-80.235,-179.798,14.784,151.050
C09738=1106.228,309.967,-80.204,-179.801,14.783,151.050
C09739=1106.223,309.718,-80.173,-179.805,14.782,151.051
C09740=1106.217,309.471,-80.142,-179.808,14.781,151.051
C09741=1106.212,309.223,-80.111,-179.812,14.779,151.052
C09742=1106.206,308.974,-80.080,-179.815,14.778,151.052
C09743=1106.200,308.727,-80.049,-179.819,14.777,151.053
C09744=1106.195,308.479,-80.018,-179.823,14.775,151.053
C09745=1106.189,308.231,-79.987,-179.826,14.775,151.054
C09746=1106.183,307.983,-79.955,-179.830,14.773,151.054
C09747=1106.177,307.735,-79.925,-179.833,14.772,151.055
C09748=1106.172,307.487,-79.894,-179.837,14.771,151.055
C09749=1106.166,307.240,-79.863,-179.840,14.770,151.056
C09750=1106.160,306.991,-79.832,-179.844,14.768,151.056
C09751=1106.154,306.743,-79.801,-179.848,14.767,151.057
C09752=1106.149,306.495,-79.770,-179.851,14.766,151.057
C09753=1106.143,306.248,-79.739,-179.855,14.764,151.058
C09754=1106.137,305.999,-79.708,-179.859,14.764,151.059
C09755=1106.132,305.751,-79.678,-179.863,14.762,151.059
C09756=1106.126,305.503,-79.646,-179.866,14.761,151.060
C09757=1106.120,305.256,-79.616,-179.870,14.760,151.060
C09758=1106.115,305.007,-79.585,-179.874,14.758,151.061
C09759=1106.109,304.759,-79.554,-179.877,14.757,151.061
C09760=1106.104,304.511,-79.523,-179.881,14.756,151.062
C09761=1106.098,304.263,-79.493,-179.884,14.755,151.062
C09762=1106.092,304.016,-79.462,-179.888,14.754,151.063
C09763=1106.087,303.768,-79.431,-179.891,14.753,151.063
C09764=1106.078,303.389,-79.384,-179.897,14.751,151.064
C09765=1106.070,303.009,-79.338,-179.903,14.750,151.065
C09766=1106.061,302.630,-79.290,-179.909,14.747,151.066
C09767=1106.052,302.251,-79.243,-179.914,14.746,151.066
C09768=1106.047,302.003,-79.213,-179.918,14.745,151.067
C09769=1106.041,301.755,-79.182,-179.921,14.744,151.068
C09770=1106.036,301.507,-79.151,-179.925,14.742,151.068
C09771=1106.030,301.259,-79.121,-179.928,14.741,151.069
C09772=1106.025,301.011,-79.090,-179.933,14.740,151.069
C09773=1106.019,300.763,-79.060,-179.936,14.739,151.070
C09774=1106.013,300.515,-79.029,-179.940,14.738,151.070
C09775=1106.008,300.267,-78.999,-179.943,14.737,151.071
C09776=1106.002,300.020,-78.968,-179.947,14.736,151.071
C09777=1105.997,299.771,-78.939,-179.950,14.735,151.072
C09778=1105.992,299.523,-78.908,-179.954,14.733,151.072
C09779=1105.986,299.275,-78.877,-179.957,14.733,151.073
C09780=1105.979,299.027,-78.847,-179.962,14.732,151.074
C09781=1105.974,298.779,-78.816,-179.965,14.731,151.074
C09782=1105.969,298.531,-78.785,-179.969,14.729,151.075
C09783=1105.963,298.283,-78.755,-179.972,14.729,151.075
C09784=1105.957,298.034,-78.725,-179.976,14.727,151.076
C09785=1105.951,297.787,-78.695,-179.980,14.727,151.076
C09786=1105.946,297.539,-78.665,-179.984,14.725,151.077
C09787=1105.940,297.291,-78.634,-179.987,14.724,151.077
C09788=1105.935,297.042,-78.604,-179.991,14.723,151.078
C09789=1105.929,296.794,-78.574,-179.994,14.722,151.079
C09790=1105.923,296.547,-78.543,-179.998,14.721,151.079
C09791=1105.917,296.299,-78.513,179.998,14.720,151.080
C09792=1105.912,296.050,-78.483,179.994,14.719,151.080
C09793=1105.906,295.802,-78.453,179.991,14.718,151.081
C09794=1105.900,295.555,-78.423,179.987,14.717,151.082
C09795=1105.895,295.306,-78.393,179.984,14.717,151.082
C09796=1105.889,295.058,-78.363,179.980,14.716,151.083
C09797=1105.884,294.810,-78.333,179.976,14.715,151.083
C09798=1105.878,294.562,-78.303,179.973,14.714,151.084
C09799=1105.872,294.314,-78.272,179.968,14.713,151.085
C09800=1105.866,294.066,-78.243,179.965,14.712,151.085
C09801=1105.861,293.818,-78.212,179.961,14.711,151.086
C09802=1105.855,293.570,-78.183,179.958,14.710,151.086
C09803=1105.849,293.322,-78.152,179.953,14.709,151.087
C09804=1105.844,293.073,-78.123,179.950,14.709,151.088
C09805=1105.838,292.825,-78.092,179.946,14.707,151.088
C09806=1105.832,292.577,-78.063,179.942,14.707,151.089
C09807=1105.827,292.329,-78.032,179.939,14.706,151.089
C09808=1105.821,292.081,-78.003,179.935,14.705,151.090
C09809=1105.815,291.833,-77.972,179.932,14.704,151.091
C09810=1105.810,291.585,-77.943,179.928,14.703,151.091
C09811=1105.804,291.337,-77.912,179.924,14.702,151.092
C09812=1105.798,291.088,-77.883,179.920,14.701,151.093
C09813=1105.793,290.840,-77.852,179.917,14.700,151.093
C09814=1105.787,290.592,-77.823,179.913,14.700,151.094
C09815=1105.782,290.344,-77.793,179.909,14.699,151.094
C09816=1105.773,289.979,-77.749,179.904,14.698,151.095
C09817=1105.764,289.614,-77.705,179.898,14.697,151.096
C09818=1105.756,289.249,-77.662,179.893,14.695,151.097
C09819=1105.748,288.884,-77.619,179.887,14.694,151.098
C09820=1105.742,288.636,-77.588,179.884,14.693,151.099
C09821=1105.737,288.387,-77.559,179.880,14.692,151.099
C09822=1105.731,288.139,-77.530,179.876,14.692,151.100
C09823=1105.725,287.891,-77.499,179.872,14.691,151.101
C09824=1105.719,287.643,-77.470,179.868,14.690,151.101
C09825=1105.714,287.395,-77.440,179.865,14.689,151.102
C09826=1105.708,287.146,-77.411,179.861,14.688,151.103
C09827=1105.702,286.898,-77.381,179.857,14.688,151.103
C09828=1105.697,286.651,-77.351,179.854,14.687,151.104
C09829=1105.691,286.402,-77.322,179.849,14.686,151.105
C09830=1105.685,286.154,-77.293,179.846,14.686,151.105
C09831=1105.680,285.906,-77.263,179.843,14.685,151.106
C09832=1105.674,285.657,-77.233,179.839,14.684,151.106
C09833=1105.668,285.409,-77.204,179.835,14.684,151.107
C09834=1105.662,285.161,-77.175,179.831,14.683,151.108
C09835=1105.657,284.913,-77.146,179.827,14.682,151.109
C09836=1105.652,284.665,-77.116,179.824,14.682,151.109
C09837=1105.646,284.417,-77.087,179.820,14.680,151.110
C09838=1105.640,284.169,-77.056,179.816,14.680,151.110
C09839=1105.634,283.920,-77.027,179.813,14.679,151.111
C09840=1105.629,283.673,-76.998,179.808,14.678,151.112
C09841=1105.623,283.424,-76.969,179.805,14.678,151.112
C09842=1105.617,283.176,-76.939,179.801,14.677,151.113
C09843=1105.611,282.928,-76.910,179.797,14.676,151.114
C09844=1105.606,282.679,-76.881,179.794,14.675,151.114
C09845=1105.600,282.431,-76.852,179.790,14.674,151.115
C09846=1105.595,282.183,-76.823,179.786,14.674,151.116
C09847=1105.589,281.934,-76.793,179.783,14.674,151.116
C09848=1105.583,281.686,-76.764,179.778,14.672,151.117
C09849=1105.578,281.439,-76.735,179.775,14.672,151.118
C09850=1105.572,281.190,-76.706,179.771,14.672,151.118
C09851=1105.567,280.942,-76.676,179.767,14.671,151.119
C09852=1105.560,280.694,-76.647,179.764,14.670,151.120
C09853=1105.556,280.446,-76.618,179.760,14.670,151.120
C09854=1105.549,280.197,-76.589,179.756,14.669,151.121
C09855=1105.544,279.949,-76.560,179.752,14.668,151.122
C09856=1105.538,279.701,-76.531,179.749,14.668,151.123
C09857=1105.533,279.453,-76.501,179.745,14.667,151.123
C09858=1105.527,279.204,-76.473,179.741,14.666,151.124
C09859=1105.521,278.956,-76.443,179.737,14.666,151.125
C09860=1105.515,278.708,-76.414,179.733,14.665,151.125
C09861=1105.509,278.460,-76.386,179.730,14.664,151.126
C09862=1105.504,278.211,-76.357,179.726,14.664,151.127
C09863=1105.498,277.963,-76.328,179.722,14.663,151.127
C09864=1105.493,277.715,-76.299,179.718,14.662,151.128
C09865=1105.487,277.467,-76.270,179.715,14.662,151.129
C09866=1105.482,277.218,-76.241,179.711,14.661,151.129
C09867=1105.476,276.971,-76.212,179.707,14.661,151.130
C09868=1105.467,276.615,-76.170,179.701,14.660,151.131
C09869=1105.459,276.259,-76.129,179.696,14.659,151.132
C09870=1105.452,275.903,-76.088,179.691,14.658,151.133
C09871=1105.443,275.548,-76.047,179.685,14.657,151.134
C09872=1105.438,275.299,-76.018,179.682,14.657,151.135
C09873=1105.432,275.051,-75.990,179.678,14.657,151.136
C09874=1105.426,274.803,-75.961,179.674,14.656,151.136
C09875=1105.421,274.554,-75.932,179.670,14.655,151.137
C09876=1105.415,274.307,-75.903,179.667,14.655,151.138
C09877=1105.409,274.058,-75.875,179.662,14.654,151.138
C09878=1105.404,273.809,-75.845,179.659,14.654,151.139
C09879=1105.398,273.561,-75.817,179.655,14.653,151.140
C09880=1105.392,273.313,-75.788,179.652,14.653,151.141
C09881=1105.386,273.064,-75.760,179.647,14.652,151.141
C09882=1105.381,272.817,-75.730,179.643,14.652,151.142
C09883=1105.375,272.568,-75.702,179.640,14.651,151.143
C09884=1105.370,272.321,-75.673,179.636,14.650,151.143
C09885=1105.364,272.072,-75.645,179.632,14.650,151.144
C09886=1105.358,271.823,-75.617,179.629,14.650,151.145
C09887=1105.352,271.576,-75.588,179.625,14.650,151.146
C09888=1105.347,271.327,-75.559,179.621,14.649,151.146
C09889=1105.341,271.078,-75.531,179.617,14.648,151.147
C09890=1105.335,270.830,-75.502,179.613,14.648,151.148
C09891=1105.330,270.582,-75.474,179.610,14.647,151.148
C09892=1105.324,270.334,-75.446,179.605,14.647,151.149
C09893=1105.318,270.085,-75.417,179.602,14.646,151.150
C09894=1105.313,269.837,-75.388,179.598,14.646,151.151
C09895=1105.307,269.588,-75.360,179.594,14.645,151.151
C09896=1105.302,269.340,-75.332,179.590,14.645,151.152
C09897=1105.296,269.092,-75.303,179.587,14.644,151.153
C09898=1105.290,268.844,-75.275,179.583,14.644,151.154
C09899=1105.284,268.595,-75.247,179.579,14.643,151.155
C09900=1105.279,268.347,-75.219,179.575,14.643,151.155
C09901=1105.273,268.099,-75.190,179.571,14.643,151.156
C09902=1105.267,267.850,-75.162,179.568,14.643,151.157
C09903=1105.261,267.602,-75.133,179.563,14.642,151.157
C09904=1105.255,267.354,-75.105,179.560,14.641,151.158
C09905=1105.250,267.106,-75.077,179.556,14.641,151.159
C09906=1105.244,266.857,-75.049,179.552,14.641,151.160
C09907=1105.239,266.609,-75.021,179.549,14.640,151.160
C09908=1105.233,266.360,-74.992,179.545,14.639,151.161
C09909=1105.228,266.112,-74.965,179.541,14.639,151.162
C09910=1105.222,265.864,-74.937,179.537,14.639,151.163
C09911=1105.216,265.615,-74.908,179.534,14.639,151.163
C09912=1105.211,265.367,-74.880,179.529,14.638,151.164
C09913=1105.205,265.118,-74.852,179.526,14.638,151.165
C09914=1105.200,264.870,-74.824,179.522,14.637,151.166
C09915=1105.194,264.622,-74.796,179.518,14.637,151.166
C09916=1105.188,264.373,-74.768,179.514,14.636,151.167
C09917=1105.182,264.125,-74.739,179.510,14.636,151.168
C09918=1105.176,263.877,-74.712,179.506,14.636,151.169
C09919=1105.170,263.628,-74.684,179.503,14.636,151.170
C09920=1105.162,263.276,-74.644,179.497,14.635,151.171
C09921=1105.154,262.923,-74.604,179.492,14.635,151.172
C09922=1105.146,262.570,-74.564,179.486,14.634,151.173
C09923=1105.138,262.217,-74.525,179.481,14.634,151.174
C09924=1105.132,261.968,-74.497,179.477,14.633,151.175
C09925=1105.127,261.720,-74.469,179.473,14.633,151.175
C09926=1105.120,261.472,-74.441,179.469,14.633,151.176
C09927=1105.115,261.224,-74.413,179.466,14.633,151.177
C09928=1105.110,260.975,-74.386,179.462,14.633,151.178
C09929=1105.103,260.727,-74.358,179.457,14.632,151.179
C09930=1105.098,260.479,-74.330,179.454,14.632,151.179
C09931=1105.092,260.230,-74.302,179.450,14.631,151.180
C09932=1105.086,259.982,-74.274,179.446,14.631,151.181
C09933=1105.081,259.733,-74.247,179.443,14.631,151.182
C09934=1105.075,259.485,-74.219,179.438,14.630,151.183
C09935=1105.069,259.237,-74.191,179.435,14.630,151.183
C09936=1105.063,258.988,-74.164,179.431,14.630,151.184
C09937=1105.058,258.740,-74.136,179.427,14.630,151.185
C09938=1105.052,258.491,-74.108,179.423,14.630,151.186
C09939=1105.046,258.242,-74.081,179.420,14.629,151.186
C09940=1105.041,257.994,-74.053,179.415,14.629,151.187
C09941=1105.035,257.746,-74.025,179.412,14.628,151.188
C09942=1105.029,257.497,-73.998,179.408,14.628,151.189
C09943=1105.023,257.249,-73.970,179.404,14.628,151.190
C09944=1105.018,257.001,-73.943,179.400,14.628,151.190
C09945=1105.012,256.752,-73.915,179.396,14.628,151.191
C09946=1105.006,256.504,-73.887,179.392,14.627,151.192
C09947=1105.001,256.256,-73.860,179.388,14.627,151.193
C09948=1104.995,256.007,-73.832,179.385,14.627,151.194
C09949=1104.990,255.758,-73.805,179.381,14.627,151.194
C09950=1104.984,255.511,-73.778,179.377,14.626,151.195
C09951=1104.978,255.261,-73.750,179.374,14.626,151.196
C09952=1104.972,255.013,-73.723,179.369,14.625,151.197
C09953=1104.967,254.765,-73.695,179.365,14.625,151.198
C09954=1104.961,254.517,-73.668,179.362,14.625,151.198
C09955=1104.955,254.268,-73.640,179.358,14.625,151.199
C09956=1104.950,254.020,-73.612,179.354,14.625,151.200
C09957=1104.944,253.771,-73.586,179.351,14.625,151.201
C09958=1104.939,253.523,-73.559,179.346,14.624,151.202
C09959=1104.932,253.274,-73.531,179.342,14.624,151.202
C09960=1104.927,253.025,-73.504,179.339,14.624,151.203
C09961=1104.921,252.777,-73.477,179.335,14.623,151.204
C09962=1104.916,252.529,-73.449,179.331,14.623,151.205
C09963=1104.910,252.280,-73.422,179.328,14.623,151.205
C09964=1104.905,252.031,-73.395,179.323,14.622,151.206
C09965=1104.899,251.784,-73.367,179.319,14.623,151.207
C09966=1104.894,251.535,-73.340,179.316,14.622,151.208
C09967=1104.888,251.287,-73.313,179.312,14.622,151.209
C09968=1104.882,251.038,-73.285,179.308,14.622,151.209
C09969=1104.876,250.789,-73.258,179.304,14.622,151.210
C09970=1104.871,250.541,-73.231,179.301,14.622,151.211
C09971=1104.865,250.292,-73.205,179.296,14.621,151.212
C09972=1104.858,249.937,-73.166,179.291,14.621,151.213
C09973=1104.849,249.582,-73.126,179.285,14.620,151.214
C09974=1104.842,249.226,-73.087,179.280,14.621,151.215
C09975=1104.833,248.870,-73.049,179.274,14.620,151.216
C09976=1104.827,248.622,-73.022,179.270,14.620,151.217
C09977=1104.822,248.373,-72.995,179.267,14.619,151.218
C09978=1104.816,248.125,-72.968,179.263,14.619,151.219
C09979=1104.811,247.876,-72.941,179.259,14.619,151.220
C09980=1104.806,247.628,-72.914,179.256,14.619,151.220
C09981=1104.800,247.379,-72.887,179.252,14.619,151.221
C09982=1104.795,247.130,-72.860,179.248,14.619,151.222
C09983=1104.789,246.882,-72.834,179.244,14.618,151.223
C09984=1104.783,246.633,-72.807,179.240,14.618,151.224
C09985=1104.777,246.385,-72.780,179.236,14.618,151.224
C09986=1104.772,246.136,-72.753,179.232,14.618,151.225
C09987=1104.766,245.888,-72.726,179.228,14.618,151.226
C09988=1104.760,245.639,-72.699,179.225,14.618,151.227
C09989=1104.755,245.391,-72.672,179.221,14.618,151.228
C09990=1104.749,245.142,-72.646,179.217,14.618,151.229
C09991=1104.744,244.894,-72.619,179.214,14.618,151.229
C09992=1104.738,244.646,-72.592,179.210,14.618,151.230
C09993=1104.732,244.397,-72.566,179.205,14.617,151.231
C09994=1104.727,244.149,-72.538,179.202,14.617,151.232
//INST
///DATE 2021/06/17 10:53
///ATTR SC,RW,RJ
////FRAME USER -1
///GROUP1 RB1
NOP
MOVJ C00000 VJ=100.00 PL=0
MOVJ C00001 VJ=100.00 PL=0
'Path Start: Op_ID_1
MOVJ C00002 VJ=25.00 PL=0
MOVJ C00003 VJ=25.00 PL=0
MOVL C00004 V=800.0 PL=0
'CALL JOB: TOOL ON
MOVL C00005 V=800.0 PL=0
MOVL C00006 V=800.0 PL=0
MOVL C00007 V=800.0 PL=0
MOVL C00008 V=800.0 PL=0
MOVL C00009 V=800.0 PL=0
MOVL C00010 V=800.0 PL=0
MOVL C00011 V=800.0 PL=0
MOVL C00012 V=800.0 PL=0
MOVL C00013 V=800.0 PL=0
MOVL C00014 V=800.0 PL=0
MOVL C00015 V=800.0 PL=0
MOVL C00016 V=800.0 PL=0
MOVL C00017 V=800.0 PL=0
MOVL C00018 V=800.0 PL=0
MOVL C00019 V=800.0 PL=0
MOVL C00020 V=800.0 PL=0
MOVL C00021 V=800.0 PL=0
MOVL C00022 V=800.0 PL=0
MOVL C00023 V=800.0 PL=0
MOVL C00024 V=800.0 PL=0
MOVL C00025 V=800.0 PL=0
MOVL C00026 V=800.0 PL=0
MOVL C00027 V=800.0 PL=0
MOVL C00028 V=800.0 PL=0
MOVL C00029 V=800.0 PL=0
MOVL C00030 V=800.0 PL=0
MOVL C00031 V=800.0 PL=0
MOVL C00032 V=800.0 PL=0
MOVL C00033 V=800.0 PL=0
MOVL C00034 V=800.0 PL=0
MOVL C00035 V=800.0 PL=0
MOVL C00036 V=800.0 PL=0
MOVL C00037 V=800.0 PL=0
MOVL C00038 V=800.0 PL=0
MOVL C00039 V=800.0 PL=0
MOVL C00040 V=800.0 PL=0
MOVL C00041 V=800.0 PL=0
MOVL C00042 V=800.0 PL=0
MOVL C00043 V=800.0 PL=0
MOVL C00044 V=800.0 PL=0
MOVL C00045 V=800.0 PL=0
MOVL C00046 V=800.0 PL=0
MOVL C00047 V=800.0 PL=0
MOVL C00048 V=800.0 PL=0
MOVL C00049 V=800.0 PL=0
MOVL C00050 V=800.0 PL=0
MOVL C00051 V=800.0 PL=0
MOVL C00052 V=800.0 PL=0
MOVL C00053 V=800.0 PL=0
MOVL C00054 V=800.0 PL=0
MOVL C00055 V=800.0 PL=0
MOVL C00056 V=800.0 PL=0
MOVL C00057 V=800.0 PL=0
MOVL C00058 V=800.0 PL=0
MOVL C00059 V=800.0 PL=0
MOVL C00060 V=800.0 PL=0
MOVL C00061 V=800.0 PL=0
MOVL C00062 V=800.0 PL=0
MOVL C00063 V=800.0 PL=0
MOVL C00064 V=800.0 PL=0
MOVL C00065 V=800.0 PL=0
MOVL C00066 V=800.0 PL=0
MOVL C00067 V=800.0 PL=0
MOVL C00068 V=800.0 PL=0
MOVL C00069 V=800.0 PL=0
MOVL C00070 V=800.0 PL=0
MOVL C00071 V=800.0 PL=0
MOVL C00072 V=800.0 PL=0
MOVL C00073 V=800.0 PL=0
MOVL C00074 V=800.0 PL=0
MOVL C00075 V=800.0 PL=0
MOVL C00076 V=800.0 PL=0
MOVL C00077 V=800.0 PL=0
MOVL C00078 V=800.0 PL=0
MOVL C00079 V=800.0 PL=0
MOVL C00080 V=800.0 PL=0
MOVL C00081 V=800.0 PL=0
MOVL C00082 V=800.0 PL=0
MOVL C00083 V=800.0 PL=0
MOVL C00084 V=800.0 PL=0
MOVL C00085 V=800.0 PL=0
MOVL C00086 V=800.0 PL=0
MOVL C00087 V=800.0 PL=0
MOVL C00088 V=800.0 PL=0
MOVL C00089 V=800.0 PL=0
MOVL C00090 V=800.0 PL=0
MOVL C00091 V=800.0 PL=0
MOVL C00092 V=800.0 PL=0
MOVL C00093 V=800.0 PL=0
MOVL C00094 V=800.0 PL=0
MOVL C00095 V=800.0 PL=0
MOVL C00096 V=800.0 PL=0
MOVL C00097 V=800.0 PL=0
MOVL C00098 V=800.0 PL=0
MOVL C00099 V=800.0 PL=0
MOVL C00100 V=800.0 PL=0
MOVL C00101 V=800.0 PL=0
MOVL C00102 V=800.0 PL=0
MOVL C00103 V=800.0 PL=0
MOVL C00104 V=800.0 PL=0
MOVL C00105 V=800.0 PL=0
MOVL C00106 V=800.0 PL=0
MOVL C00107 V=800.0 PL=0
MOVL C00108 V=800.0 PL=0
MOVL C00109 V=800.0 PL=0
MOVL C00110 V=800.0 PL=0
MOVL C00111 V=800.0 PL=0
MOVL C00112 V=800.0 PL=0
MOVL C00113 V=800.0 PL=0
MOVL C00114 V=800.0 PL=0
MOVL C00115 V=800.0 PL=0
MOVL C00116 V=800.0 PL=0
MOVL C00117 V=800.0 PL=0
MOVL C00118 V=800.0 PL=0
MOVL C00119 V=800.0 PL=0
MOVL C00120 V=800.0 PL=0
MOVL C00121 V=800.0 PL=0
MOVL C00122 V=800.0 PL=0
MOVL C00123 V=800.0 PL=0
MOVL C00124 V=800.0 PL=0
MOVL C00125 V=800.0 PL=0
MOVL C00126 V=800.0 PL=0
MOVL C00127 V=800.0 PL=0
MOVL C00128 V=800.0 PL=0
MOVL C00129 V=800.0 PL=0
MOVL C00130 V=800.0 PL=0
MOVL C00131 V=800.0 PL=0
MOVL C00132 V=800.0 PL=0
MOVL C00133 V=800.0 PL=0
MOVL C00134 V=800.0 PL=0
MOVL C00135 V=800.0 PL=0
MOVL C00136 V=800.0 PL=0
MOVL C00137 V=800.0 PL=0
MOVL C00138 V=800.0 PL=0
MOVL C00139 V=800.0 PL=0
MOVL C00140 V=800.0 PL=0
MOVL C00141 V=800.0 PL=0
MOVL C00142 V=800.0 PL=0
MOVL C00143 V=800.0 PL=0
MOVL C00144 V=800.0 PL=0
MOVL C00145 V=800.0 PL=0
MOVL C00146 V=800.0 PL=0
MOVL C00147 V=800.0 PL=0
MOVL C00148 V=800.0 PL=0
MOVL C00149 V=800.0 PL=0
MOVL C00150 V=800.0 PL=0
MOVL C00151 V=800.0 PL=0
MOVL C00152 V=800.0 PL=0
MOVL C00153 V=800.0 PL=0
MOVL C00154 V=800.0 PL=0
MOVL C00155 V=800.0 PL=0
MOVL C00156 V=800.0 PL=0
MOVL C00157 V=800.0 PL=0
MOVL C00158 V=800.0 PL=0
MOVL C00159 V=800.0 PL=0
MOVL C00160 V=800.0 PL=0
MOVL C00161 V=800.0 PL=0
MOVL C00162 V=800.0 PL=0
MOVL C00163 V=800.0 PL=0
MOVL C00164 V=800.0 PL=0
MOVL C00165 V=800.0 PL=0
MOVL C00166 V=800.0 PL=0
MOVL C00167 V=800.0 PL=0
MOVL C00168 V=800.0 PL=0
MOVL C00169 V=800.0 PL=0
MOVL C00170 V=800.0 PL=0
MOVL C00171 V=800.0 PL=0
MOVL C00172 V=800.0 PL=0
MOVL C00173 V=800.0 PL=0
MOVL C00174 V=800.0 PL=0
MOVL C00175 V=800.0 PL=0
MOVL C00176 V=800.0 PL=0
MOVL C00177 V=800.0 PL=0
MOVL C00178 V=800.0 PL=0
MOVL C00179 V=800.0 PL=0
MOVL C00180 V=800.0 PL=0
MOVL C00181 V=800.0 PL=0
MOVL C00182 V=800.0 PL=0
MOVL C00183 V=800.0 PL=0
MOVL C00184 V=800.0 PL=0
MOVL C00185 V=800.0 PL=0
MOVL C00186 V=800.0 PL=0
MOVL C00187 V=800.0 PL=0
MOVL C00188 V=800.0 PL=0
MOVL C00189 V=800.0 PL=0
MOVL C00190 V=800.0 PL=0
MOVL C00191 V=800.0 PL=0
MOVL C00192 V=800.0 PL=0
MOVL C00193 V=800.0 PL=0
MOVL C00194 V=800.0 PL=0
MOVL C00195 V=800.0 PL=0
MOVL C00196 V=800.0 PL=0
MOVL C00197 V=800.0 PL=0
MOVL C00198 V=800.0 PL=0
MOVL C00199 V=800.0 PL=0
MOVL C00200 V=800.0 PL=0
MOVL C00201 V=800.0 PL=0
MOVL C00202 V=800.0 PL=0
MOVL C00203 V=800.0 PL=0
MOVL C00204 V=800.0 PL=0
MOVL C00205 V=800.0 PL=0
MOVL C00206 V=800.0 PL=0
MOVL C00207 V=800.0 PL=0
MOVL C00208 V=800.0 PL=0
MOVL C00209 V=800.0 PL=0
MOVL C00210 V=800.0 PL=0
MOVL C00211 V=800.0 PL=0
MOVL C00212 V=800.0 PL=0
MOVL C00213 V=800.0 PL=0
MOVL C00214 V=800.0 PL=0
MOVL C00215 V=800.0 PL=0
MOVL C00216 V=800.0 PL=0
MOVL C00217 V=800.0 PL=0
MOVL C00218 V=800.0 PL=0
MOVL C00219 V=800.0 PL=0
MOVL C00220 V=800.0 PL=0
MOVL C00221 V=800.0 PL=0
MOVL C00222 V=800.0 PL=0
MOVL C00223 V=800.0 PL=0
MOVL C00224 V=800.0 PL=0
MOVL C00225 V=800.0 PL=0
MOVL C00226 V=800.0 PL=0
MOVL C00227 V=800.0 PL=0
MOVL C00228 V=800.0 PL=0
MOVL C00229 V=800.0 PL=0
MOVL C00230 V=800.0 PL=0
MOVL C00231 V=800.0 PL=0
MOVL C00232 V=800.0 PL=0
MOVL C00233 V=800.0 PL=0
MOVL C00234 V=800.0 PL=0
MOVL C00235 V=800.0 PL=0
MOVL C00236 V=800.0 PL=0
MOVL C00237 V=800.0 PL=0
MOVL C00238 V=800.0 PL=0
MOVL C00239 V=800.0 PL=0
MOVL C00240 V=800.0 PL=0
MOVL C00241 V=800.0 PL=0
MOVL C00242 V=800.0 PL=0
MOVL C00243 V=800.0 PL=0
MOVL C00244 V=800.0 PL=0
MOVL C00245 V=800.0 PL=0
MOVL C00246 V=800.0 PL=0
MOVL C00247 V=800.0 PL=0
MOVL C00248 V=800.0 PL=0
MOVL C00249 V=800.0 PL=0
MOVL C00250 V=800.0 PL=0
MOVL C00251 V=800.0 PL=0
MOVL C00252 V=800.0 PL=0
MOVL C00253 V=800.0 PL=0
MOVL C00254 V=800.0 PL=0
MOVL C00255 V=800.0 PL=0
MOVL C00256 V=800.0 PL=0
MOVL C00257 V=800.0 PL=0
MOVL C00258 V=800.0 PL=0
MOVL C00259 V=800.0 PL=0
MOVL C00260 V=800.0 PL=0
MOVL C00261 V=800.0 PL=0
MOVL C00262 V=800.0 PL=0
MOVL C00263 V=800.0 PL=0
MOVL C00264 V=800.0 PL=0
MOVL C00265 V=800.0 PL=0
MOVL C00266 V=800.0 PL=0
MOVL C00267 V=800.0 PL=0
MOVL C00268 V=800.0 PL=0
MOVL C00269 V=800.0 PL=0
MOVL C00270 V=800.0 PL=0
MOVL C00271 V=800.0 PL=0
MOVL C00272 V=800.0 PL=0
MOVL C00273 V=800.0 PL=0
MOVL C00274 V=800.0 PL=0
MOVL C00275 V=800.0 PL=0
MOVL C00276 V=800.0 PL=0
MOVL C00277 V=800.0 PL=0
MOVL C00278 V=800.0 PL=0
MOVL C00279 V=800.0 PL=0
MOVL C00280 V=800.0 PL=0
MOVL C00281 V=800.0 PL=0
MOVL C00282 V=800.0 PL=0
MOVL C00283 V=800.0 PL=0
MOVL C00284 V=800.0 PL=0
MOVL C00285 V=800.0 PL=0
MOVL C00286 V=800.0 PL=0
MOVL C00287 V=800.0 PL=0
MOVL C00288 V=800.0 PL=0
MOVL C00289 V=800.0 PL=0
MOVL C00290 V=800.0 PL=0
MOVL C00291 V=800.0 PL=0
MOVL C00292 V=800.0 PL=0
MOVL C00293 V=800.0 PL=0
MOVL C00294 V=800.0 PL=0
MOVL C00295 V=800.0 PL=0
MOVL C00296 V=800.0 PL=0
MOVL C00297 V=800.0 PL=0
MOVL C00298 V=800.0 PL=0
MOVL C00299 V=800.0 PL=0
MOVL C00300 V=800.0 PL=0
MOVL C00301 V=800.0 PL=0
MOVL C00302 V=800.0 PL=0
MOVL C00303 V=800.0 PL=0
MOVL C00304 V=800.0 PL=0
MOVL C00305 V=800.0 PL=0
MOVL C00306 V=800.0 PL=0
MOVL C00307 V=800.0 PL=0
MOVL C00308 V=800.0 PL=0
MOVL C00309 V=800.0 PL=0
MOVL C00310 V=800.0 PL=0
MOVL C00311 V=800.0 PL=0
MOVL C00312 V=800.0 PL=0
MOVL C00313 V=800.0 PL=0
MOVL C00314 V=800.0 PL=0
MOVL C00315 V=800.0 PL=0
MOVL C00316 V=800.0 PL=0
MOVL C00317 V=800.0 PL=0
MOVL C00318 V=800.0 PL=0
MOVL C00319 V=800.0 PL=0
MOVL C00320 V=800.0 PL=0
MOVL C00321 V=800.0 PL=0
MOVL C00322 V=800.0 PL=0
MOVL C00323 V=800.0 PL=0
MOVL C00324 V=800.0 PL=0
MOVL C00325 V=800.0 PL=0
MOVL C00326 V=800.0 PL=0
MOVL C00327 V=800.0 PL=0
MOVL C00328 V=800.0 PL=0
MOVL C00329 V=800.0 PL=0
MOVL C00330 V=800.0 PL=0
MOVL C00331 V=800.0 PL=0
MOVL C00332 V=800.0 PL=0
MOVL C00333 V=800.0 PL=0
MOVL C00334 V=800.0 PL=0
MOVL C00335 V=800.0 PL=0
MOVL C00336 V=800.0 PL=0
MOVL C00337 V=800.0 PL=0
MOVL C00338 V=800.0 PL=0
MOVL C00339 V=800.0 PL=0
MOVL C00340 V=800.0 PL=0
MOVL C00341 V=800.0 PL=0
MOVL C00342 V=800.0 PL=0
MOVL C00343 V=800.0 PL=0
MOVL C00344 V=800.0 PL=0
MOVL C00345 V=800.0 PL=0
MOVL C00346 V=800.0 PL=0
MOVL C00347 V=800.0 PL=0
MOVL C00348 V=800.0 PL=0
MOVL C00349 V=800.0 PL=0
MOVL C00350 V=800.0 PL=0
MOVL C00351 V=800.0 PL=0
MOVL C00352 V=800.0 PL=0
MOVL C00353 V=800.0 PL=0
MOVL C00354 V=800.0 PL=0
MOVL C00355 V=800.0 PL=0
MOVL C00356 V=800.0 PL=0
MOVL C00357 V=800.0 PL=0
MOVL C00358 V=800.0 PL=0
MOVL C00359 V=800.0 PL=0
MOVL C00360 V=800.0 PL=0
MOVL C00361 V=800.0 PL=0
MOVL C00362 V=800.0 PL=0
MOVL C00363 V=800.0 PL=0
MOVL C00364 V=800.0 PL=0
MOVL C00365 V=800.0 PL=0
MOVL C00366 V=800.0 PL=0
MOVL C00367 V=800.0 PL=0
MOVL C00368 V=800.0 PL=0
MOVL C00369 V=800.0 PL=0
MOVL C00370 V=800.0 PL=0
MOVL C00371 V=800.0 PL=0
MOVL C00372 V=800.0 PL=0
MOVL C00373 V=800.0 PL=0
MOVL C00374 V=800.0 PL=0
MOVL C00375 V=800.0 PL=0
MOVL C00376 V=800.0 PL=0
MOVL C00377 V=800.0 PL=0
MOVL C00378 V=800.0 PL=0
MOVL C00379 V=800.0 PL=0
MOVL C00380 V=800.0 PL=0
MOVL C00381 V=800.0 PL=0
MOVL C00382 V=800.0 PL=0
MOVL C00383 V=800.0 PL=0
MOVL C00384 V=800.0 PL=0
MOVL C00385 V=800.0 PL=0
MOVL C00386 V=800.0 PL=0
MOVL C00387 V=800.0 PL=0
MOVL C00388 V=800.0 PL=0
MOVL C00389 V=800.0 PL=0
MOVL C00390 V=800.0 PL=0
MOVL C00391 V=800.0 PL=0
MOVL C00392 V=800.0 PL=0
MOVL C00393 V=800.0 PL=0
MOVL C00394 V=800.0 PL=0
MOVL C00395 V=800.0 PL=0
MOVL C00396 V=800.0 PL=0
MOVL C00397 V=800.0 PL=0
MOVL C00398 V=800.0 PL=0
MOVL C00399 V=800.0 PL=0
MOVL C00400 V=800.0 PL=0
MOVL C00401 V=800.0 PL=0
MOVL C00402 V=800.0 PL=0
MOVL C00403 V=800.0 PL=0
MOVL C00404 V=800.0 PL=0
MOVL C00405 V=800.0 PL=0
MOVL C00406 V=800.0 PL=0
MOVL C00407 V=800.0 PL=0
MOVL C00408 V=800.0 PL=0
MOVL C00409 V=800.0 PL=0
MOVL C00410 V=800.0 PL=0
MOVL C00411 V=800.0 PL=0
MOVL C00412 V=800.0 PL=0
MOVL C00413 V=800.0 PL=0
MOVL C00414 V=800.0 PL=0
MOVL C00415 V=800.0 PL=0
MOVL C00416 V=800.0 PL=0
MOVL C00417 V=800.0 PL=0
MOVL C00418 V=800.0 PL=0
MOVL C00419 V=800.0 PL=0
MOVL C00420 V=800.0 PL=0
MOVL C00421 V=800.0 PL=0
MOVL C00422 V=800.0 PL=0
MOVL C00423 V=800.0 PL=0
MOVL C00424 V=800.0 PL=0
MOVL C00425 V=800.0 PL=0
MOVL C00426 V=800.0 PL=0
MOVL C00427 V=800.0 PL=0
MOVL C00428 V=800.0 PL=0
MOVL C00429 V=800.0 PL=0
MOVL C00430 V=800.0 PL=0
MOVL C00431 V=800.0 PL=0
MOVL C00432 V=800.0 PL=0
MOVL C00433 V=800.0 PL=0
MOVL C00434 V=800.0 PL=0
MOVL C00435 V=800.0 PL=0
MOVL C00436 V=800.0 PL=0
MOVL C00437 V=800.0 PL=0
MOVL C00438 V=800.0 PL=0
MOVL C00439 V=800.0 PL=0
MOVL C00440 V=800.0 PL=0
MOVL C00441 V=800.0 PL=0
MOVL C00442 V=800.0 PL=0
MOVL C00443 V=800.0 PL=0
MOVL C00444 V=800.0 PL=0
MOVL C00445 V=800.0 PL=0
MOVL C00446 V=800.0 PL=0
MOVL C00447 V=800.0 PL=0
MOVL C00448 V=800.0 PL=0
MOVL C00449 V=800.0 PL=0
MOVL C00450 V=800.0 PL=0
MOVL C00451 V=800.0 PL=0
MOVL C00452 V=800.0 PL=0
MOVL C00453 V=800.0 PL=0
MOVL C00454 V=800.0 PL=0
MOVL C00455 V=800.0 PL=0
MOVL C00456 V=800.0 PL=0
MOVL C00457 V=800.0 PL=0
MOVL C00458 V=800.0 PL=0
MOVL C00459 V=800.0 PL=0
MOVL C00460 V=800.0 PL=0
MOVL C00461 V=800.0 PL=0
MOVL C00462 V=800.0 PL=0
MOVL C00463 V=800.0 PL=0
MOVL C00464 V=800.0 PL=0
MOVL C00465 V=800.0 PL=0
MOVL C00466 V=800.0 PL=0
MOVL C00467 V=800.0 PL=0
MOVL C00468 V=800.0 PL=0
MOVL C00469 V=800.0 PL=0
MOVL C00470 V=800.0 PL=0
MOVL C00471 V=800.0 PL=0
MOVL C00472 V=800.0 PL=0
MOVL C00473 V=800.0 PL=0
MOVL C00474 V=800.0 PL=0
MOVL C00475 V=800.0 PL=0
MOVL C00476 V=800.0 PL=0
MOVL C00477 V=800.0 PL=0
MOVL C00478 V=800.0 PL=0
MOVL C00479 V=800.0 PL=0
MOVL C00480 V=800.0 PL=0
MOVL C00481 V=800.0 PL=0
MOVL C00482 V=800.0 PL=0
MOVL C00483 V=800.0 PL=0
MOVL C00484 V=800.0 PL=0
MOVL C00485 V=800.0 PL=0
MOVL C00486 V=800.0 PL=0
MOVL C00487 V=800.0 PL=0
MOVL C00488 V=800.0 PL=0
MOVL C00489 V=800.0 PL=0
MOVL C00490 V=800.0 PL=0
MOVL C00491 V=800.0 PL=0
MOVL C00492 V=800.0 PL=0
MOVL C00493 V=800.0 PL=0
MOVL C00494 V=800.0 PL=0
MOVL C00495 V=800.0 PL=0
MOVL C00496 V=800.0 PL=0
MOVL C00497 V=800.0 PL=0
MOVL C00498 V=800.0 PL=0
MOVL C00499 V=800.0 PL=0
MOVL C00500 V=800.0 PL=0
MOVL C00501 V=800.0 PL=0
MOVL C00502 V=800.0 PL=0
MOVL C00503 V=800.0 PL=0
MOVL C00504 V=800.0 PL=0
MOVL C00505 V=800.0 PL=0
MOVL C00506 V=800.0 PL=0
MOVL C00507 V=800.0 PL=0
MOVL C00508 V=800.0 PL=0
MOVL C00509 V=800.0 PL=0
MOVL C00510 V=800.0 PL=0
MOVL C00511 V=800.0 PL=0
MOVL C00512 V=800.0 PL=0
MOVL C00513 V=800.0 PL=0
MOVL C00514 V=800.0 PL=0
MOVL C00515 V=800.0 PL=0
MOVL C00516 V=800.0 PL=0
MOVL C00517 V=800.0 PL=0
MOVL C00518 V=800.0 PL=0
MOVL C00519 V=800.0 PL=0
MOVL C00520 V=800.0 PL=0
MOVL C00521 V=800.0 PL=0
MOVL C00522 V=800.0 PL=0
MOVL C00523 V=800.0 PL=0
MOVL C00524 V=800.0 PL=0
MOVL C00525 V=800.0 PL=0
MOVL C00526 V=800.0 PL=0
MOVL C00527 V=800.0 PL=0
MOVL C00528 V=800.0 PL=0
MOVL C00529 V=800.0 PL=0
MOVL C00530 V=800.0 PL=0
MOVL C00531 V=800.0 PL=0
MOVL C00532 V=800.0 PL=0
MOVL C00533 V=800.0 PL=0
MOVL C00534 V=800.0 PL=0
MOVL C00535 V=800.0 PL=0
MOVL C00536 V=800.0 PL=0
MOVL C00537 V=800.0 PL=0
MOVL C00538 V=800.0 PL=0
MOVL C00539 V=800.0 PL=0
MOVL C00540 V=800.0 PL=0
MOVL C00541 V=800.0 PL=0
MOVL C00542 V=800.0 PL=0
MOVL C00543 V=800.0 PL=0
MOVL C00544 V=800.0 PL=0
MOVL C00545 V=800.0 PL=0
MOVL C00546 V=800.0 PL=0
MOVL C00547 V=800.0 PL=0
MOVL C00548 V=800.0 PL=0
MOVL C00549 V=800.0 PL=0
MOVL C00550 V=800.0 PL=0
MOVL C00551 V=800.0 PL=0
MOVL C00552 V=800.0 PL=0
MOVL C00553 V=800.0 PL=0
MOVL C00554 V=800.0 PL=0
MOVL C00555 V=800.0 PL=0
MOVL C00556 V=800.0 PL=0
MOVL C00557 V=800.0 PL=0
MOVL C00558 V=800.0 PL=0
MOVL C00559 V=800.0 PL=0
MOVL C00560 V=800.0 PL=0
MOVL C00561 V=800.0 PL=0
MOVL C00562 V=800.0 PL=0
MOVL C00563 V=800.0 PL=0
MOVL C00564 V=800.0 PL=0
MOVL C00565 V=800.0 PL=0
MOVL C00566 V=800.0 PL=0
MOVL C00567 V=800.0 PL=0
MOVL C00568 V=800.0 PL=0
MOVL C00569 V=800.0 PL=0
MOVL C00570 V=800.0 PL=0
MOVL C00571 V=800.0 PL=0
MOVL C00572 V=800.0 PL=0
MOVL C00573 V=800.0 PL=0
MOVL C00574 V=800.0 PL=0
MOVL C00575 V=800.0 PL=0
MOVL C00576 V=800.0 PL=0
MOVL C00577 V=800.0 PL=0
MOVL C00578 V=800.0 PL=0
MOVL C00579 V=800.0 PL=0
MOVL C00580 V=800.0 PL=0
MOVL C00581 V=800.0 PL=0
MOVL C00582 V=800.0 PL=0
MOVL C00583 V=800.0 PL=0
MOVL C00584 V=800.0 PL=0
MOVL C00585 V=800.0 PL=0
MOVL C00586 V=800.0 PL=0
MOVL C00587 V=800.0 PL=0
MOVL C00588 V=800.0 PL=0
MOVL C00589 V=800.0 PL=0
MOVL C00590 V=800.0 PL=0
MOVL C00591 V=800.0 PL=0
MOVL C00592 V=800.0 PL=0
MOVL C00593 V=800.0 PL=0
MOVL C00594 V=800.0 PL=0
MOVL C00595 V=800.0 PL=0
MOVL C00596 V=800.0 PL=0
MOVL C00597 V=800.0 PL=0
MOVL C00598 V=800.0 PL=0
MOVL C00599 V=800.0 PL=0
MOVL C00600 V=800.0 PL=0
MOVL C00601 V=800.0 PL=0
MOVL C00602 V=800.0 PL=0
MOVL C00603 V=800.0 PL=0
MOVL C00604 V=800.0 PL=0
MOVL C00605 V=800.0 PL=0
MOVL C00606 V=800.0 PL=0
MOVL C00607 V=800.0 PL=0
MOVL C00608 V=800.0 PL=0
MOVL C00609 V=800.0 PL=0
MOVL C00610 V=800.0 PL=0
MOVL C00611 V=800.0 PL=0
MOVL C00612 V=800.0 PL=0
MOVL C00613 V=800.0 PL=0
MOVL C00614 V=800.0 PL=0
MOVL C00615 V=800.0 PL=0
MOVL C00616 V=800.0 PL=0
MOVL C00617 V=800.0 PL=0
MOVL C00618 V=800.0 PL=0
MOVL C00619 V=800.0 PL=0
MOVL C00620 V=800.0 PL=0
MOVL C00621 V=800.0 PL=0
MOVL C00622 V=800.0 PL=0
MOVL C00623 V=800.0 PL=0
MOVL C00624 V=800.0 PL=0
MOVL C00625 V=800.0 PL=0
MOVL C00626 V=800.0 PL=0
MOVL C00627 V=800.0 PL=0
MOVL C00628 V=800.0 PL=0
MOVL C00629 V=800.0 PL=0
MOVL C00630 V=800.0 PL=0
MOVL C00631 V=800.0 PL=0
MOVL C00632 V=800.0 PL=0
MOVL C00633 V=800.0 PL=0
MOVL C00634 V=800.0 PL=0
MOVL C00635 V=800.0 PL=0
MOVL C00636 V=800.0 PL=0
MOVL C00637 V=800.0 PL=0
MOVL C00638 V=800.0 PL=0
MOVL C00639 V=800.0 PL=0
MOVL C00640 V=800.0 PL=0
MOVL C00641 V=800.0 PL=0
MOVL C00642 V=800.0 PL=0
MOVL C00643 V=800.0 PL=0
MOVL C00644 V=800.0 PL=0
MOVL C00645 V=800.0 PL=0
MOVL C00646 V=800.0 PL=0
MOVL C00647 V=800.0 PL=0
MOVL C00648 V=800.0 PL=0
MOVL C00649 V=800.0 PL=0
MOVL C00650 V=800.0 PL=0
MOVL C00651 V=800.0 PL=0
MOVL C00652 V=800.0 PL=0
MOVL C00653 V=800.0 PL=0
MOVL C00654 V=800.0 PL=0
MOVL C00655 V=800.0 PL=0
MOVL C00656 V=800.0 PL=0
MOVL C00657 V=800.0 PL=0
MOVL C00658 V=800.0 PL=0
MOVL C00659 V=800.0 PL=0
MOVL C00660 V=800.0 PL=0
MOVL C00661 V=800.0 PL=0
MOVL C00662 V=800.0 PL=0
MOVL C00663 V=800.0 PL=0
MOVL C00664 V=800.0 PL=0
MOVL C00665 V=800.0 PL=0
MOVL C00666 V=800.0 PL=0
MOVL C00667 V=800.0 PL=0
MOVL C00668 V=800.0 PL=0
MOVL C00669 V=800.0 PL=0
MOVL C00670 V=800.0 PL=0
MOVL C00671 V=800.0 PL=0
MOVL C00672 V=800.0 PL=0
MOVL C00673 V=800.0 PL=0
MOVL C00674 V=800.0 PL=0
MOVL C00675 V=800.0 PL=0
MOVL C00676 V=800.0 PL=0
MOVL C00677 V=800.0 PL=0
MOVL C00678 V=800.0 PL=0
MOVL C00679 V=800.0 PL=0
MOVL C00680 V=800.0 PL=0
MOVL C00681 V=800.0 PL=0
MOVL C00682 V=800.0 PL=0
MOVL C00683 V=800.0 PL=0
MOVL C00684 V=800.0 PL=0
MOVL C00685 V=800.0 PL=0
MOVL C00686 V=800.0 PL=0
MOVL C00687 V=800.0 PL=0
MOVL C00688 V=800.0 PL=0
MOVL C00689 V=800.0 PL=0
MOVL C00690 V=800.0 PL=0
MOVL C00691 V=800.0 PL=0
MOVL C00692 V=800.0 PL=0
MOVL C00693 V=800.0 PL=0
MOVL C00694 V=800.0 PL=0
MOVL C00695 V=800.0 PL=0
MOVL C00696 V=800.0 PL=0
MOVL C00697 V=800.0 PL=0
MOVL C00698 V=800.0 PL=0
MOVL C00699 V=800.0 PL=0
MOVL C00700 V=800.0 PL=0
MOVL C00701 V=800.0 PL=0
MOVL C00702 V=800.0 PL=0
MOVL C00703 V=800.0 PL=0
MOVL C00704 V=800.0 PL=0
MOVL C00705 V=800.0 PL=0
MOVL C00706 V=800.0 PL=0
MOVL C00707 V=800.0 PL=0
MOVL C00708 V=800.0 PL=0
MOVL C00709 V=800.0 PL=0
MOVL C00710 V=800.0 PL=0
MOVL C00711 V=800.0 PL=0
MOVL C00712 V=800.0 PL=0
MOVL C00713 V=800.0 PL=0
MOVL C00714 V=800.0 PL=0
MOVL C00715 V=800.0 PL=0
MOVL C00716 V=800.0 PL=0
MOVL C00717 V=800.0 PL=0
MOVL C00718 V=800.0 PL=0
MOVL C00719 V=800.0 PL=0
MOVL C00720 V=800.0 PL=0
MOVL C00721 V=800.0 PL=0
MOVL C00722 V=800.0 PL=0
MOVL C00723 V=800.0 PL=0
MOVL C00724 V=800.0 PL=0
MOVL C00725 V=800.0 PL=0
MOVL C00726 V=800.0 PL=0
MOVL C00727 V=800.0 PL=0
MOVL C00728 V=800.0 PL=0
MOVL C00729 V=800.0 PL=0
MOVL C00730 V=800.0 PL=0
MOVL C00731 V=800.0 PL=0
MOVL C00732 V=800.0 PL=0
MOVL C00733 V=800.0 PL=0
MOVL C00734 V=800.0 PL=0
MOVL C00735 V=800.0 PL=0
MOVL C00736 V=800.0 PL=0
MOVL C00737 V=800.0 PL=0
MOVL C00738 V=800.0 PL=0
MOVL C00739 V=800.0 PL=0
MOVL C00740 V=800.0 PL=0
MOVL C00741 V=800.0 PL=0
MOVL C00742 V=800.0 PL=0
MOVL C00743 V=800.0 PL=0
MOVL C00744 V=800.0 PL=0
MOVL C00745 V=800.0 PL=0
MOVL C00746 V=800.0 PL=0
MOVL C00747 V=800.0 PL=0
MOVL C00748 V=800.0 PL=0
MOVL C00749 V=800.0 PL=0
MOVL C00750 V=800.0 PL=0
MOVL C00751 V=800.0 PL=0
MOVL C00752 V=800.0 PL=0
MOVL C00753 V=800.0 PL=0
MOVL C00754 V=800.0 PL=0
MOVL C00755 V=800.0 PL=0
MOVL C00756 V=800.0 PL=0
MOVL C00757 V=800.0 PL=0
MOVL C00758 V=800.0 PL=0
MOVL C00759 V=800.0 PL=0
MOVL C00760 V=800.0 PL=0
MOVL C00761 V=800.0 PL=0
MOVL C00762 V=800.0 PL=0
MOVL C00763 V=800.0 PL=0
MOVL C00764 V=800.0 PL=0
MOVL C00765 V=800.0 PL=0
MOVL C00766 V=800.0 PL=0
MOVL C00767 V=800.0 PL=0
MOVL C00768 V=800.0 PL=0
MOVL C00769 V=800.0 PL=0
MOVL C00770 V=800.0 PL=0
MOVL C00771 V=800.0 PL=0
MOVL C00772 V=800.0 PL=0
MOVL C00773 V=800.0 PL=0
MOVL C00774 V=800.0 PL=0
MOVL C00775 V=800.0 PL=0
MOVL C00776 V=800.0 PL=0
MOVL C00777 V=800.0 PL=0
MOVL C00778 V=800.0 PL=0
MOVL C00779 V=800.0 PL=0
MOVL C00780 V=800.0 PL=0
MOVL C00781 V=800.0 PL=0
MOVL C00782 V=800.0 PL=0
MOVL C00783 V=800.0 PL=0
MOVL C00784 V=800.0 PL=0
MOVL C00785 V=800.0 PL=0
MOVL C00786 V=800.0 PL=0
MOVL C00787 V=800.0 PL=0
MOVL C00788 V=800.0 PL=0
MOVL C00789 V=800.0 PL=0
MOVL C00790 V=800.0 PL=0
MOVL C00791 V=800.0 PL=0
MOVL C00792 V=800.0 PL=0
MOVL C00793 V=800.0 PL=0
MOVL C00794 V=800.0 PL=0
MOVL C00795 V=800.0 PL=0
MOVL C00796 V=800.0 PL=0
MOVL C00797 V=800.0 PL=0
MOVL C00798 V=800.0 PL=0
MOVL C00799 V=800.0 PL=0
MOVL C00800 V=800.0 PL=0
MOVL C00801 V=800.0 PL=0
MOVL C00802 V=800.0 PL=0
MOVL C00803 V=800.0 PL=0
MOVL C00804 V=800.0 PL=0
MOVL C00805 V=800.0 PL=0
MOVL C00806 V=800.0 PL=0
MOVL C00807 V=800.0 PL=0
MOVL C00808 V=800.0 PL=0
MOVL C00809 V=800.0 PL=0
MOVL C00810 V=800.0 PL=0
MOVL C00811 V=800.0 PL=0
MOVL C00812 V=800.0 PL=0
MOVL C00813 V=800.0 PL=0
MOVL C00814 V=800.0 PL=0
MOVL C00815 V=800.0 PL=0
MOVL C00816 V=800.0 PL=0
MOVL C00817 V=800.0 PL=0
MOVL C00818 V=800.0 PL=0
MOVL C00819 V=800.0 PL=0
MOVL C00820 V=800.0 PL=0
MOVL C00821 V=800.0 PL=0
MOVL C00822 V=800.0 PL=0
MOVL C00823 V=800.0 PL=0
MOVL C00824 V=800.0 PL=0
MOVL C00825 V=800.0 PL=0
MOVL C00826 V=800.0 PL=0
MOVL C00827 V=800.0 PL=0
MOVL C00828 V=800.0 PL=0
MOVL C00829 V=800.0 PL=0
MOVL C00830 V=800.0 PL=0
MOVL C00831 V=800.0 PL=0
MOVL C00832 V=800.0 PL=0
MOVL C00833 V=800.0 PL=0
MOVL C00834 V=800.0 PL=0
MOVL C00835 V=800.0 PL=0
MOVL C00836 V=800.0 PL=0
MOVL C00837 V=800.0 PL=0
MOVL C00838 V=800.0 PL=0
MOVL C00839 V=800.0 PL=0
MOVL C00840 V=800.0 PL=0
MOVL C00841 V=800.0 PL=0
MOVL C00842 V=800.0 PL=0
MOVL C00843 V=800.0 PL=0
MOVL C00844 V=800.0 PL=0
MOVL C00845 V=800.0 PL=0
MOVL C00846 V=800.0 PL=0
MOVL C00847 V=800.0 PL=0
MOVL C00848 V=800.0 PL=0
MOVL C00849 V=800.0 PL=0
MOVL C00850 V=800.0 PL=0
MOVL C00851 V=800.0 PL=0
MOVL C00852 V=800.0 PL=0
MOVL C00853 V=800.0 PL=0
MOVL C00854 V=800.0 PL=0
MOVL C00855 V=800.0 PL=0
MOVL C00856 V=800.0 PL=0
MOVL C00857 V=800.0 PL=0
MOVL C00858 V=800.0 PL=0
MOVL C00859 V=800.0 PL=0
MOVL C00860 V=800.0 PL=0
MOVL C00861 V=800.0 PL=0
MOVL C00862 V=800.0 PL=0
MOVL C00863 V=800.0 PL=0
MOVL C00864 V=800.0 PL=0
MOVL C00865 V=800.0 PL=0
MOVL C00866 V=800.0 PL=0
MOVL C00867 V=800.0 PL=0
MOVL C00868 V=800.0 PL=0
MOVL C00869 V=800.0 PL=0
MOVL C00870 V=800.0 PL=0
MOVL C00871 V=800.0 PL=0
MOVL C00872 V=800.0 PL=0
MOVL C00873 V=800.0 PL=0
MOVL C00874 V=800.0 PL=0
MOVL C00875 V=800.0 PL=0
MOVL C00876 V=800.0 PL=0
MOVL C00877 V=800.0 PL=0
MOVL C00878 V=800.0 PL=0
MOVL C00879 V=800.0 PL=0
MOVL C00880 V=800.0 PL=0
MOVL C00881 V=800.0 PL=0
MOVL C00882 V=800.0 PL=0
MOVL C00883 V=800.0 PL=0
MOVL C00884 V=800.0 PL=0
MOVL C00885 V=800.0 PL=0
MOVL C00886 V=800.0 PL=0
MOVL C00887 V=800.0 PL=0
MOVL C00888 V=800.0 PL=0
MOVL C00889 V=800.0 PL=0
MOVL C00890 V=800.0 PL=0
MOVL C00891 V=800.0 PL=0
MOVL C00892 V=800.0 PL=0
MOVL C00893 V=800.0 PL=0
MOVL C00894 V=800.0 PL=0
MOVL C00895 V=800.0 PL=0
MOVL C00896 V=800.0 PL=0
MOVL C00897 V=800.0 PL=0
MOVL C00898 V=800.0 PL=0
MOVL C00899 V=800.0 PL=0
MOVL C00900 V=800.0 PL=0
MOVL C00901 V=800.0 PL=0
MOVL C00902 V=800.0 PL=0
MOVL C00903 V=800.0 PL=0
MOVL C00904 V=800.0 PL=0
MOVL C00905 V=800.0 PL=0
MOVL C00906 V=800.0 PL=0
MOVL C00907 V=800.0 PL=0
MOVL C00908 V=800.0 PL=0
MOVL C00909 V=800.0 PL=0
MOVL C00910 V=800.0 PL=0
MOVL C00911 V=800.0 PL=0
MOVL C00912 V=800.0 PL=0
MOVL C00913 V=800.0 PL=0
MOVL C00914 V=800.0 PL=0
MOVL C00915 V=800.0 PL=0
MOVL C00916 V=800.0 PL=0
MOVL C00917 V=800.0 PL=0
MOVL C00918 V=800.0 PL=0
MOVL C00919 V=800.0 PL=0
MOVL C00920 V=800.0 PL=0
MOVL C00921 V=800.0 PL=0
MOVL C00922 V=800.0 PL=0
MOVL C00923 V=800.0 PL=0
MOVL C00924 V=800.0 PL=0
MOVL C00925 V=800.0 PL=0
MOVL C00926 V=800.0 PL=0
MOVL C00927 V=800.0 PL=0
MOVL C00928 V=800.0 PL=0
MOVL C00929 V=800.0 PL=0
MOVL C00930 V=800.0 PL=0
MOVL C00931 V=800.0 PL=0
MOVL C00932 V=800.0 PL=0
MOVL C00933 V=800.0 PL=0
MOVL C00934 V=800.0 PL=0
MOVL C00935 V=800.0 PL=0
MOVL C00936 V=800.0 PL=0
MOVL C00937 V=800.0 PL=0
MOVL C00938 V=800.0 PL=0
MOVL C00939 V=800.0 PL=0
MOVL C00940 V=800.0 PL=0
MOVL C00941 V=800.0 PL=0
MOVL C00942 V=800.0 PL=0
MOVL C00943 V=800.0 PL=0
MOVL C00944 V=800.0 PL=0
MOVL C00945 V=800.0 PL=0
MOVL C00946 V=800.0 PL=0
MOVL C00947 V=800.0 PL=0
MOVL C00948 V=800.0 PL=0
MOVL C00949 V=800.0 PL=0
MOVL C00950 V=800.0 PL=0
MOVL C00951 V=800.0 PL=0
MOVL C00952 V=800.0 PL=0
MOVL C00953 V=800.0 PL=0
MOVL C00954 V=800.0 PL=0
MOVL C00955 V=800.0 PL=0
MOVL C00956 V=800.0 PL=0
MOVL C00957 V=800.0 PL=0
MOVL C00958 V=800.0 PL=0
MOVL C00959 V=800.0 PL=0
MOVL C00960 V=800.0 PL=0
MOVL C00961 V=800.0 PL=0
MOVL C00962 V=800.0 PL=0
MOVL C00963 V=800.0 PL=0
MOVL C00964 V=800.0 PL=0
MOVL C00965 V=800.0 PL=0
MOVL C00966 V=800.0 PL=0
MOVL C00967 V=800.0 PL=0
MOVL C00968 V=800.0 PL=0
MOVL C00969 V=800.0 PL=0
MOVL C00970 V=800.0 PL=0
MOVL C00971 V=800.0 PL=0
MOVL C00972 V=800.0 PL=0
MOVL C00973 V=800.0 PL=0
MOVL C00974 V=800.0 PL=0
MOVL C00975 V=800.0 PL=0
MOVL C00976 V=800.0 PL=0
MOVL C00977 V=800.0 PL=0
MOVL C00978 V=800.0 PL=0
MOVL C00979 V=800.0 PL=0
MOVL C00980 V=800.0 PL=0
MOVL C00981 V=800.0 PL=0
MOVL C00982 V=800.0 PL=0
MOVL C00983 V=800.0 PL=0
MOVL C00984 V=800.0 PL=0
MOVL C00985 V=800.0 PL=0
MOVL C00986 V=800.0 PL=0
MOVL C00987 V=800.0 PL=0
MOVL C00988 V=800.0 PL=0
MOVL C00989 V=800.0 PL=0
MOVL C00990 V=800.0 PL=0
MOVL C00991 V=800.0 PL=0
MOVL C00992 V=800.0 PL=0
MOVL C00993 V=800.0 PL=0
MOVL C00994 V=800.0 PL=0
MOVL C00995 V=800.0 PL=0
MOVL C00996 V=800.0 PL=0
MOVL C00997 V=800.0 PL=0
MOVL C00998 V=800.0 PL=0
MOVL C00999 V=800.0 PL=0
MOVL C01000 V=800.0 PL=0
MOVL C01001 V=800.0 PL=0
MOVL C01002 V=800.0 PL=0
MOVL C01003 V=800.0 PL=0
MOVL C01004 V=800.0 PL=0
MOVL C01005 V=800.0 PL=0
MOVL C01006 V=800.0 PL=0
MOVL C01007 V=800.0 PL=0
MOVL C01008 V=800.0 PL=0
MOVL C01009 V=800.0 PL=0
MOVL C01010 V=800.0 PL=0
MOVL C01011 V=800.0 PL=0
MOVL C01012 V=800.0 PL=0
MOVL C01013 V=800.0 PL=0
MOVL C01014 V=800.0 PL=0
MOVL C01015 V=800.0 PL=0
MOVL C01016 V=800.0 PL=0
MOVL C01017 V=800.0 PL=0
MOVL C01018 V=800.0 PL=0
MOVL C01019 V=800.0 PL=0
MOVL C01020 V=800.0 PL=0
MOVL C01021 V=800.0 PL=0
MOVL C01022 V=800.0 PL=0
MOVL C01023 V=800.0 PL=0
MOVL C01024 V=800.0 PL=0
MOVL C01025 V=800.0 PL=0
MOVL C01026 V=800.0 PL=0
MOVL C01027 V=800.0 PL=0
MOVL C01028 V=800.0 PL=0
MOVL C01029 V=800.0 PL=0
MOVL C01030 V=800.0 PL=0
MOVL C01031 V=800.0 PL=0
MOVL C01032 V=800.0 PL=0
MOVL C01033 V=800.0 PL=0
MOVL C01034 V=800.0 PL=0
MOVL C01035 V=800.0 PL=0
MOVL C01036 V=800.0 PL=0
MOVL C01037 V=800.0 PL=0
MOVL C01038 V=800.0 PL=0
MOVL C01039 V=800.0 PL=0
MOVL C01040 V=800.0 PL=0
MOVL C01041 V=800.0 PL=0
MOVL C01042 V=800.0 PL=0
MOVL C01043 V=800.0 PL=0
MOVL C01044 V=800.0 PL=0
MOVL C01045 V=800.0 PL=0
MOVL C01046 V=800.0 PL=0
MOVL C01047 V=800.0 PL=0
MOVL C01048 V=800.0 PL=0
MOVL C01049 V=800.0 PL=0
MOVL C01050 V=800.0 PL=0
MOVL C01051 V=800.0 PL=0
MOVL C01052 V=800.0 PL=0
MOVL C01053 V=800.0 PL=0
MOVL C01054 V=800.0 PL=0
MOVL C01055 V=800.0 PL=0
MOVL C01056 V=800.0 PL=0
MOVL C01057 V=800.0 PL=0
MOVL C01058 V=800.0 PL=0
MOVL C01059 V=800.0 PL=0
MOVL C01060 V=800.0 PL=0
MOVL C01061 V=800.0 PL=0
MOVL C01062 V=800.0 PL=0
MOVL C01063 V=800.0 PL=0
MOVL C01064 V=800.0 PL=0
MOVL C01065 V=800.0 PL=0
MOVL C01066 V=800.0 PL=0
MOVL C01067 V=800.0 PL=0
MOVL C01068 V=800.0 PL=0
MOVL C01069 V=800.0 PL=0
MOVL C01070 V=800.0 PL=0
MOVL C01071 V=800.0 PL=0
MOVL C01072 V=800.0 PL=0
MOVL C01073 V=800.0 PL=0
MOVL C01074 V=800.0 PL=0
MOVL C01075 V=800.0 PL=0
MOVL C01076 V=800.0 PL=0
MOVL C01077 V=800.0 PL=0
MOVL C01078 V=800.0 PL=0
MOVL C01079 V=800.0 PL=0
MOVL C01080 V=800.0 PL=0
MOVL C01081 V=800.0 PL=0
MOVL C01082 V=800.0 PL=0
MOVL C01083 V=800.0 PL=0
MOVL C01084 V=800.0 PL=0
MOVL C01085 V=800.0 PL=0
MOVL C01086 V=800.0 PL=0
MOVL C01087 V=800.0 PL=0
MOVL C01088 V=800.0 PL=0
MOVL C01089 V=800.0 PL=0
MOVL C01090 V=800.0 PL=0
MOVL C01091 V=800.0 PL=0
MOVL C01092 V=800.0 PL=0
MOVL C01093 V=800.0 PL=0
MOVL C01094 V=800.0 PL=0
MOVL C01095 V=800.0 PL=0
MOVL C01096 V=800.0 PL=0
MOVL C01097 V=800.0 PL=0
MOVL C01098 V=800.0 PL=0
MOVL C01099 V=800.0 PL=0
MOVL C01100 V=800.0 PL=0
MOVL C01101 V=800.0 PL=0
MOVL C01102 V=800.0 PL=0
MOVL C01103 V=800.0 PL=0
MOVL C01104 V=800.0 PL=0
MOVL C01105 V=800.0 PL=0
MOVL C01106 V=800.0 PL=0
MOVL C01107 V=800.0 PL=0
MOVL C01108 V=800.0 PL=0
MOVL C01109 V=800.0 PL=0
MOVL C01110 V=800.0 PL=0
MOVL C01111 V=800.0 PL=0
MOVL C01112 V=800.0 PL=0
MOVL C01113 V=800.0 PL=0
MOVL C01114 V=800.0 PL=0
MOVL C01115 V=800.0 PL=0
MOVL C01116 V=800.0 PL=0
MOVL C01117 V=800.0 PL=0
MOVL C01118 V=800.0 PL=0
MOVL C01119 V=800.0 PL=0
MOVL C01120 V=800.0 PL=0
MOVL C01121 V=800.0 PL=0
MOVL C01122 V=800.0 PL=0
MOVL C01123 V=800.0 PL=0
MOVL C01124 V=800.0 PL=0
MOVL C01125 V=800.0 PL=0
MOVL C01126 V=800.0 PL=0
MOVL C01127 V=800.0 PL=0
MOVL C01128 V=800.0 PL=0
MOVL C01129 V=800.0 PL=0
MOVL C01130 V=800.0 PL=0
MOVL C01131 V=800.0 PL=0
MOVL C01132 V=800.0 PL=0
MOVL C01133 V=800.0 PL=0
MOVL C01134 V=800.0 PL=0
MOVL C01135 V=800.0 PL=0
MOVL C01136 V=800.0 PL=0
MOVL C01137 V=800.0 PL=0
MOVL C01138 V=800.0 PL=0
MOVL C01139 V=800.0 PL=0
MOVL C01140 V=800.0 PL=0
MOVL C01141 V=800.0 PL=0
MOVL C01142 V=800.0 PL=0
MOVL C01143 V=800.0 PL=0
MOVL C01144 V=800.0 PL=0
MOVL C01145 V=800.0 PL=0
MOVL C01146 V=800.0 PL=0
MOVL C01147 V=800.0 PL=0
MOVL C01148 V=800.0 PL=0
MOVL C01149 V=800.0 PL=0
MOVL C01150 V=800.0 PL=0
MOVL C01151 V=800.0 PL=0
MOVL C01152 V=800.0 PL=0
MOVL C01153 V=800.0 PL=0
MOVL C01154 V=800.0 PL=0
MOVL C01155 V=800.0 PL=0
MOVL C01156 V=800.0 PL=0
MOVL C01157 V=800.0 PL=0
MOVL C01158 V=800.0 PL=0
MOVL C01159 V=800.0 PL=0
MOVL C01160 V=800.0 PL=0
MOVL C01161 V=800.0 PL=0
MOVL C01162 V=800.0 PL=0
MOVL C01163 V=800.0 PL=0
MOVL C01164 V=800.0 PL=0
MOVL C01165 V=800.0 PL=0
MOVL C01166 V=800.0 PL=0
MOVL C01167 V=800.0 PL=0
MOVL C01168 V=800.0 PL=0
MOVL C01169 V=800.0 PL=0
MOVL C01170 V=800.0 PL=0
MOVL C01171 V=800.0 PL=0
MOVL C01172 V=800.0 PL=0
MOVL C01173 V=800.0 PL=0
MOVL C01174 V=800.0 PL=0
MOVL C01175 V=800.0 PL=0
MOVL C01176 V=800.0 PL=0
MOVL C01177 V=800.0 PL=0
MOVL C01178 V=800.0 PL=0
MOVL C01179 V=800.0 PL=0
MOVL C01180 V=800.0 PL=0
MOVL C01181 V=800.0 PL=0
MOVL C01182 V=800.0 PL=0
MOVL C01183 V=800.0 PL=0
MOVL C01184 V=800.0 PL=0
MOVL C01185 V=800.0 PL=0
MOVL C01186 V=800.0 PL=0
MOVL C01187 V=800.0 PL=0
MOVL C01188 V=800.0 PL=0
MOVL C01189 V=800.0 PL=0
MOVL C01190 V=800.0 PL=0
MOVL C01191 V=800.0 PL=0
MOVL C01192 V=800.0 PL=0
MOVL C01193 V=800.0 PL=0
MOVL C01194 V=800.0 PL=0
MOVL C01195 V=800.0 PL=0
MOVL C01196 V=800.0 PL=0
MOVL C01197 V=800.0 PL=0
MOVL C01198 V=800.0 PL=0
MOVL C01199 V=800.0 PL=0
MOVL C01200 V=800.0 PL=0
MOVL C01201 V=800.0 PL=0
MOVL C01202 V=800.0 PL=0
MOVL C01203 V=800.0 PL=0
MOVL C01204 V=800.0 PL=0
MOVL C01205 V=800.0 PL=0
MOVL C01206 V=800.0 PL=0
MOVL C01207 V=800.0 PL=0
MOVL C01208 V=800.0 PL=0
MOVL C01209 V=800.0 PL=0
MOVL C01210 V=800.0 PL=0
MOVL C01211 V=800.0 PL=0
MOVL C01212 V=800.0 PL=0
MOVL C01213 V=800.0 PL=0
MOVL C01214 V=800.0 PL=0
MOVL C01215 V=800.0 PL=0
MOVL C01216 V=800.0 PL=0
MOVL C01217 V=800.0 PL=0
MOVL C01218 V=800.0 PL=0
MOVL C01219 V=800.0 PL=0
MOVL C01220 V=800.0 PL=0
MOVL C01221 V=800.0 PL=0
MOVL C01222 V=800.0 PL=0
MOVL C01223 V=800.0 PL=0
MOVL C01224 V=800.0 PL=0
MOVL C01225 V=800.0 PL=0
MOVL C01226 V=800.0 PL=0
MOVL C01227 V=800.0 PL=0
MOVL C01228 V=800.0 PL=0
MOVL C01229 V=800.0 PL=0
MOVL C01230 V=800.0 PL=0
MOVL C01231 V=800.0 PL=0
MOVL C01232 V=800.0 PL=0
MOVL C01233 V=800.0 PL=0
MOVL C01234 V=800.0 PL=0
MOVL C01235 V=800.0 PL=0
MOVL C01236 V=800.0 PL=0
MOVL C01237 V=800.0 PL=0
MOVL C01238 V=800.0 PL=0
MOVL C01239 V=800.0 PL=0
MOVL C01240 V=800.0 PL=0
MOVL C01241 V=800.0 PL=0
MOVL C01242 V=800.0 PL=0
MOVL C01243 V=800.0 PL=0
MOVL C01244 V=800.0 PL=0
MOVL C01245 V=800.0 PL=0
MOVL C01246 V=800.0 PL=0
MOVL C01247 V=800.0 PL=0
MOVL C01248 V=800.0 PL=0
MOVL C01249 V=800.0 PL=0
MOVL C01250 V=800.0 PL=0
MOVL C01251 V=800.0 PL=0
MOVL C01252 V=800.0 PL=0
MOVL C01253 V=800.0 PL=0
MOVL C01254 V=800.0 PL=0
MOVL C01255 V=800.0 PL=0
MOVL C01256 V=800.0 PL=0
MOVL C01257 V=800.0 PL=0
MOVL C01258 V=800.0 PL=0
MOVL C01259 V=800.0 PL=0
MOVL C01260 V=800.0 PL=0
MOVL C01261 V=800.0 PL=0
MOVL C01262 V=800.0 PL=0
MOVL C01263 V=800.0 PL=0
MOVL C01264 V=800.0 PL=0
MOVL C01265 V=800.0 PL=0
MOVL C01266 V=800.0 PL=0
MOVL C01267 V=800.0 PL=0
MOVL C01268 V=800.0 PL=0
MOVL C01269 V=800.0 PL=0
MOVL C01270 V=800.0 PL=0
MOVL C01271 V=800.0 PL=0
MOVL C01272 V=800.0 PL=0
MOVL C01273 V=800.0 PL=0
MOVL C01274 V=800.0 PL=0
MOVL C01275 V=800.0 PL=0
MOVL C01276 V=800.0 PL=0
MOVL C01277 V=800.0 PL=0
MOVL C01278 V=800.0 PL=0
MOVL C01279 V=800.0 PL=0
MOVL C01280 V=800.0 PL=0
MOVL C01281 V=800.0 PL=0
MOVL C01282 V=800.0 PL=0
MOVL C01283 V=800.0 PL=0
MOVL C01284 V=800.0 PL=0
MOVL C01285 V=800.0 PL=0
MOVL C01286 V=800.0 PL=0
MOVL C01287 V=800.0 PL=0
MOVL C01288 V=800.0 PL=0
MOVL C01289 V=800.0 PL=0
MOVL C01290 V=800.0 PL=0
MOVL C01291 V=800.0 PL=0
MOVL C01292 V=800.0 PL=0
MOVL C01293 V=800.0 PL=0
MOVL C01294 V=800.0 PL=0
MOVL C01295 V=800.0 PL=0
MOVL C01296 V=800.0 PL=0
MOVL C01297 V=800.0 PL=0
MOVL C01298 V=800.0 PL=0
MOVL C01299 V=800.0 PL=0
MOVL C01300 V=800.0 PL=0
MOVL C01301 V=800.0 PL=0
MOVL C01302 V=800.0 PL=0
MOVL C01303 V=800.0 PL=0
MOVL C01304 V=800.0 PL=0
MOVL C01305 V=800.0 PL=0
MOVL C01306 V=800.0 PL=0
MOVL C01307 V=800.0 PL=0
MOVL C01308 V=800.0 PL=0
MOVL C01309 V=800.0 PL=0
MOVL C01310 V=800.0 PL=0
MOVL C01311 V=800.0 PL=0
MOVL C01312 V=800.0 PL=0
MOVL C01313 V=800.0 PL=0
MOVL C01314 V=800.0 PL=0
MOVL C01315 V=800.0 PL=0
MOVL C01316 V=800.0 PL=0
MOVL C01317 V=800.0 PL=0
MOVL C01318 V=800.0 PL=0
MOVL C01319 V=800.0 PL=0
MOVL C01320 V=800.0 PL=0
MOVL C01321 V=800.0 PL=0
MOVL C01322 V=800.0 PL=0
MOVL C01323 V=800.0 PL=0
MOVL C01324 V=800.0 PL=0
MOVL C01325 V=800.0 PL=0
MOVL C01326 V=800.0 PL=0
MOVL C01327 V=800.0 PL=0
MOVL C01328 V=800.0 PL=0
MOVL C01329 V=800.0 PL=0
MOVL C01330 V=800.0 PL=0
MOVL C01331 V=800.0 PL=0
MOVL C01332 V=800.0 PL=0
MOVL C01333 V=800.0 PL=0
MOVL C01334 V=800.0 PL=0
MOVL C01335 V=800.0 PL=0
MOVL C01336 V=800.0 PL=0
MOVL C01337 V=800.0 PL=0
MOVL C01338 V=800.0 PL=0
MOVL C01339 V=800.0 PL=0
MOVL C01340 V=800.0 PL=0
MOVL C01341 V=800.0 PL=0
MOVL C01342 V=800.0 PL=0
MOVL C01343 V=800.0 PL=0
MOVL C01344 V=800.0 PL=0
MOVL C01345 V=800.0 PL=0
MOVL C01346 V=800.0 PL=0
MOVL C01347 V=800.0 PL=0
MOVL C01348 V=800.0 PL=0
MOVL C01349 V=800.0 PL=0
MOVL C01350 V=800.0 PL=0
MOVL C01351 V=800.0 PL=0
MOVL C01352 V=800.0 PL=0
MOVL C01353 V=800.0 PL=0
MOVL C01354 V=800.0 PL=0
MOVL C01355 V=800.0 PL=0
MOVL C01356 V=800.0 PL=0
MOVL C01357 V=800.0 PL=0
MOVL C01358 V=800.0 PL=0
MOVL C01359 V=800.0 PL=0
MOVL C01360 V=800.0 PL=0
MOVL C01361 V=800.0 PL=0
MOVL C01362 V=800.0 PL=0
MOVL C01363 V=800.0 PL=0
MOVL C01364 V=800.0 PL=0
MOVL C01365 V=800.0 PL=0
MOVL C01366 V=800.0 PL=0
MOVL C01367 V=800.0 PL=0
MOVL C01368 V=800.0 PL=0
MOVL C01369 V=800.0 PL=0
MOVL C01370 V=800.0 PL=0
MOVL C01371 V=800.0 PL=0
MOVL C01372 V=800.0 PL=0
MOVL C01373 V=800.0 PL=0
MOVL C01374 V=800.0 PL=0
MOVL C01375 V=800.0 PL=0
MOVL C01376 V=800.0 PL=0
MOVL C01377 V=800.0 PL=0
MOVL C01378 V=800.0 PL=0
MOVL C01379 V=800.0 PL=0
MOVL C01380 V=800.0 PL=0
MOVL C01381 V=800.0 PL=0
MOVL C01382 V=800.0 PL=0
MOVL C01383 V=800.0 PL=0
MOVL C01384 V=800.0 PL=0
MOVL C01385 V=800.0 PL=0
MOVL C01386 V=800.0 PL=0
MOVL C01387 V=800.0 PL=0
MOVL C01388 V=800.0 PL=0
MOVL C01389 V=800.0 PL=0
MOVL C01390 V=800.0 PL=0
MOVL C01391 V=800.0 PL=0
MOVL C01392 V=800.0 PL=0
MOVL C01393 V=800.0 PL=0
MOVL C01394 V=800.0 PL=0
MOVL C01395 V=800.0 PL=0
MOVL C01396 V=800.0 PL=0
MOVL C01397 V=800.0 PL=0
MOVL C01398 V=800.0 PL=0
MOVL C01399 V=800.0 PL=0
MOVL C01400 V=800.0 PL=0
MOVL C01401 V=800.0 PL=0
MOVL C01402 V=800.0 PL=0
MOVL C01403 V=800.0 PL=0
MOVL C01404 V=800.0 PL=0
MOVL C01405 V=800.0 PL=0
MOVL C01406 V=800.0 PL=0
MOVL C01407 V=800.0 PL=0
MOVL C01408 V=800.0 PL=0
MOVL C01409 V=800.0 PL=0
MOVL C01410 V=800.0 PL=0
MOVL C01411 V=800.0 PL=0
MOVL C01412 V=800.0 PL=0
MOVL C01413 V=800.0 PL=0
MOVL C01414 V=800.0 PL=0
MOVL C01415 V=800.0 PL=0
MOVL C01416 V=800.0 PL=0
MOVL C01417 V=800.0 PL=0
MOVL C01418 V=800.0 PL=0
MOVL C01419 V=800.0 PL=0
MOVL C01420 V=800.0 PL=0
MOVL C01421 V=800.0 PL=0
MOVL C01422 V=800.0 PL=0
MOVL C01423 V=800.0 PL=0
MOVL C01424 V=800.0 PL=0
MOVL C01425 V=800.0 PL=0
MOVL C01426 V=800.0 PL=0
MOVL C01427 V=800.0 PL=0
MOVL C01428 V=800.0 PL=0
MOVL C01429 V=800.0 PL=0
MOVL C01430 V=800.0 PL=0
MOVL C01431 V=800.0 PL=0
MOVL C01432 V=800.0 PL=0
MOVL C01433 V=800.0 PL=0
MOVL C01434 V=800.0 PL=0
MOVL C01435 V=800.0 PL=0
MOVL C01436 V=800.0 PL=0
MOVL C01437 V=800.0 PL=0
MOVL C01438 V=800.0 PL=0
MOVL C01439 V=800.0 PL=0
MOVL C01440 V=800.0 PL=0
MOVL C01441 V=800.0 PL=0
MOVL C01442 V=800.0 PL=0
MOVL C01443 V=800.0 PL=0
MOVL C01444 V=800.0 PL=0
MOVL C01445 V=800.0 PL=0
MOVL C01446 V=800.0 PL=0
MOVL C01447 V=800.0 PL=0
MOVL C01448 V=800.0 PL=0
MOVL C01449 V=800.0 PL=0
MOVL C01450 V=800.0 PL=0
MOVL C01451 V=800.0 PL=0
MOVL C01452 V=800.0 PL=0
MOVL C01453 V=800.0 PL=0
MOVL C01454 V=800.0 PL=0
MOVL C01455 V=800.0 PL=0
MOVL C01456 V=800.0 PL=0
MOVL C01457 V=800.0 PL=0
MOVL C01458 V=800.0 PL=0
MOVL C01459 V=800.0 PL=0
MOVL C01460 V=800.0 PL=0
MOVL C01461 V=800.0 PL=0
MOVL C01462 V=800.0 PL=0
MOVL C01463 V=800.0 PL=0
MOVL C01464 V=800.0 PL=0
MOVL C01465 V=800.0 PL=0
MOVL C01466 V=800.0 PL=0
MOVL C01467 V=800.0 PL=0
MOVL C01468 V=800.0 PL=0
MOVL C01469 V=800.0 PL=0
MOVL C01470 V=800.0 PL=0
MOVL C01471 V=800.0 PL=0
MOVL C01472 V=800.0 PL=0
MOVL C01473 V=800.0 PL=0
MOVL C01474 V=800.0 PL=0
MOVL C01475 V=800.0 PL=0
MOVL C01476 V=800.0 PL=0
MOVL C01477 V=800.0 PL=0
MOVL C01478 V=800.0 PL=0
MOVL C01479 V=800.0 PL=0
MOVL C01480 V=800.0 PL=0
MOVL C01481 V=800.0 PL=0
MOVL C01482 V=800.0 PL=0
MOVL C01483 V=800.0 PL=0
MOVL C01484 V=800.0 PL=0
MOVL C01485 V=800.0 PL=0
MOVL C01486 V=800.0 PL=0
MOVL C01487 V=800.0 PL=0
MOVL C01488 V=800.0 PL=0
MOVL C01489 V=800.0 PL=0
MOVL C01490 V=800.0 PL=0
MOVL C01491 V=800.0 PL=0
MOVL C01492 V=800.0 PL=0
MOVL C01493 V=800.0 PL=0
MOVL C01494 V=800.0 PL=0
MOVL C01495 V=800.0 PL=0
MOVL C01496 V=800.0 PL=0
MOVL C01497 V=800.0 PL=0
MOVL C01498 V=800.0 PL=0
MOVL C01499 V=800.0 PL=0
MOVL C01500 V=800.0 PL=0
MOVL C01501 V=800.0 PL=0
MOVL C01502 V=800.0 PL=0
MOVL C01503 V=800.0 PL=0
MOVL C01504 V=800.0 PL=0
MOVL C01505 V=800.0 PL=0
MOVL C01506 V=800.0 PL=0
MOVL C01507 V=800.0 PL=0
MOVL C01508 V=800.0 PL=0
MOVL C01509 V=800.0 PL=0
MOVL C01510 V=800.0 PL=0
MOVL C01511 V=800.0 PL=0
MOVL C01512 V=800.0 PL=0
MOVL C01513 V=800.0 PL=0
MOVL C01514 V=800.0 PL=0
MOVL C01515 V=800.0 PL=0
MOVL C01516 V=800.0 PL=0
MOVL C01517 V=800.0 PL=0
MOVL C01518 V=800.0 PL=0
MOVL C01519 V=800.0 PL=0
MOVL C01520 V=800.0 PL=0
MOVL C01521 V=800.0 PL=0
MOVL C01522 V=800.0 PL=0
MOVL C01523 V=800.0 PL=0
MOVL C01524 V=800.0 PL=0
MOVL C01525 V=800.0 PL=0
MOVL C01526 V=800.0 PL=0
MOVL C01527 V=800.0 PL=0
MOVL C01528 V=800.0 PL=0
MOVL C01529 V=800.0 PL=0
MOVL C01530 V=800.0 PL=0
MOVL C01531 V=800.0 PL=0
MOVL C01532 V=800.0 PL=0
MOVL C01533 V=800.0 PL=0
MOVL C01534 V=800.0 PL=0
MOVL C01535 V=800.0 PL=0
MOVL C01536 V=800.0 PL=0
MOVL C01537 V=800.0 PL=0
MOVL C01538 V=800.0 PL=0
MOVL C01539 V=800.0 PL=0
MOVL C01540 V=800.0 PL=0
MOVL C01541 V=800.0 PL=0
MOVL C01542 V=800.0 PL=0
MOVL C01543 V=800.0 PL=0
MOVL C01544 V=800.0 PL=0
MOVL C01545 V=800.0 PL=0
MOVL C01546 V=800.0 PL=0
MOVL C01547 V=800.0 PL=0
MOVL C01548 V=800.0 PL=0
MOVL C01549 V=800.0 PL=0
MOVL C01550 V=800.0 PL=0
MOVL C01551 V=800.0 PL=0
MOVL C01552 V=800.0 PL=0
MOVL C01553 V=800.0 PL=0
MOVL C01554 V=800.0 PL=0
MOVL C01555 V=800.0 PL=0
MOVL C01556 V=800.0 PL=0
MOVL C01557 V=800.0 PL=0
MOVL C01558 V=800.0 PL=0
MOVL C01559 V=800.0 PL=0
MOVL C01560 V=800.0 PL=0
MOVL C01561 V=800.0 PL=0
MOVL C01562 V=800.0 PL=0
MOVL C01563 V=800.0 PL=0
MOVL C01564 V=800.0 PL=0
MOVL C01565 V=800.0 PL=0
MOVL C01566 V=800.0 PL=0
MOVL C01567 V=800.0 PL=0
MOVL C01568 V=800.0 PL=0
MOVL C01569 V=800.0 PL=0
MOVL C01570 V=800.0 PL=0
MOVL C01571 V=800.0 PL=0
MOVL C01572 V=800.0 PL=0
MOVL C01573 V=800.0 PL=0
MOVL C01574 V=800.0 PL=0
MOVL C01575 V=800.0 PL=0
MOVL C01576 V=800.0 PL=0
MOVL C01577 V=800.0 PL=0
MOVL C01578 V=800.0 PL=0
MOVL C01579 V=800.0 PL=0
MOVL C01580 V=800.0 PL=0
MOVL C01581 V=800.0 PL=0
MOVL C01582 V=800.0 PL=0
MOVL C01583 V=800.0 PL=0
MOVL C01584 V=800.0 PL=0
MOVL C01585 V=800.0 PL=0
MOVL C01586 V=800.0 PL=0
MOVL C01587 V=800.0 PL=0
MOVL C01588 V=800.0 PL=0
MOVL C01589 V=800.0 PL=0
MOVL C01590 V=800.0 PL=0
MOVL C01591 V=800.0 PL=0
MOVL C01592 V=800.0 PL=0
MOVL C01593 V=800.0 PL=0
MOVL C01594 V=800.0 PL=0
MOVL C01595 V=800.0 PL=0
MOVL C01596 V=800.0 PL=0
MOVL C01597 V=800.0 PL=0
MOVL C01598 V=800.0 PL=0
MOVL C01599 V=800.0 PL=0
MOVL C01600 V=800.0 PL=0
MOVL C01601 V=800.0 PL=0
MOVL C01602 V=800.0 PL=0
MOVL C01603 V=800.0 PL=0
MOVL C01604 V=800.0 PL=0
MOVL C01605 V=800.0 PL=0
MOVL C01606 V=800.0 PL=0
MOVL C01607 V=800.0 PL=0
MOVL C01608 V=800.0 PL=0
MOVL C01609 V=800.0 PL=0
MOVL C01610 V=800.0 PL=0
MOVL C01611 V=800.0 PL=0
MOVL C01612 V=800.0 PL=0
MOVL C01613 V=800.0 PL=0
MOVL C01614 V=800.0 PL=0
MOVL C01615 V=800.0 PL=0
MOVL C01616 V=800.0 PL=0
MOVL C01617 V=800.0 PL=0
MOVL C01618 V=800.0 PL=0
MOVL C01619 V=800.0 PL=0
MOVL C01620 V=800.0 PL=0
MOVL C01621 V=800.0 PL=0
MOVL C01622 V=800.0 PL=0
MOVL C01623 V=800.0 PL=0
MOVL C01624 V=800.0 PL=0
MOVL C01625 V=800.0 PL=0
MOVL C01626 V=800.0 PL=0
MOVL C01627 V=800.0 PL=0
MOVL C01628 V=800.0 PL=0
MOVL C01629 V=800.0 PL=0
MOVL C01630 V=800.0 PL=0
MOVL C01631 V=800.0 PL=0
MOVL C01632 V=800.0 PL=0
MOVL C01633 V=800.0 PL=0
MOVL C01634 V=800.0 PL=0
MOVL C01635 V=800.0 PL=0
MOVL C01636 V=800.0 PL=0
MOVL C01637 V=800.0 PL=0
MOVL C01638 V=800.0 PL=0
MOVL C01639 V=800.0 PL=0
MOVL C01640 V=800.0 PL=0
MOVL C01641 V=800.0 PL=0
MOVL C01642 V=800.0 PL=0
MOVL C01643 V=800.0 PL=0
MOVL C01644 V=800.0 PL=0
MOVL C01645 V=800.0 PL=0
MOVL C01646 V=800.0 PL=0
MOVL C01647 V=800.0 PL=0
MOVL C01648 V=800.0 PL=0
MOVL C01649 V=800.0 PL=0
MOVL C01650 V=800.0 PL=0
MOVL C01651 V=800.0 PL=0
MOVL C01652 V=800.0 PL=0
MOVL C01653 V=800.0 PL=0
MOVL C01654 V=800.0 PL=0
MOVL C01655 V=800.0 PL=0
MOVL C01656 V=800.0 PL=0
MOVL C01657 V=800.0 PL=0
MOVL C01658 V=800.0 PL=0
MOVL C01659 V=800.0 PL=0
MOVL C01660 V=800.0 PL=0
MOVL C01661 V=800.0 PL=0
MOVL C01662 V=800.0 PL=0
MOVL C01663 V=800.0 PL=0
MOVL C01664 V=800.0 PL=0
MOVL C01665 V=800.0 PL=0
MOVL C01666 V=800.0 PL=0
MOVL C01667 V=800.0 PL=0
MOVL C01668 V=800.0 PL=0
MOVL C01669 V=800.0 PL=0
MOVL C01670 V=800.0 PL=0
MOVL C01671 V=800.0 PL=0
MOVL C01672 V=800.0 PL=0
MOVL C01673 V=800.0 PL=0
MOVL C01674 V=800.0 PL=0
MOVL C01675 V=800.0 PL=0
MOVL C01676 V=800.0 PL=0
MOVL C01677 V=800.0 PL=0
MOVL C01678 V=800.0 PL=0
MOVL C01679 V=800.0 PL=0
MOVL C01680 V=800.0 PL=0
MOVL C01681 V=800.0 PL=0
MOVL C01682 V=800.0 PL=0
MOVL C01683 V=800.0 PL=0
MOVL C01684 V=800.0 PL=0
MOVL C01685 V=800.0 PL=0
MOVL C01686 V=800.0 PL=0
MOVL C01687 V=800.0 PL=0
MOVL C01688 V=800.0 PL=0
MOVL C01689 V=800.0 PL=0
MOVL C01690 V=800.0 PL=0
MOVL C01691 V=800.0 PL=0
MOVL C01692 V=800.0 PL=0
MOVL C01693 V=800.0 PL=0
MOVL C01694 V=800.0 PL=0
MOVL C01695 V=800.0 PL=0
MOVL C01696 V=800.0 PL=0
MOVL C01697 V=800.0 PL=0
MOVL C01698 V=800.0 PL=0
MOVL C01699 V=800.0 PL=0
MOVL C01700 V=800.0 PL=0
MOVL C01701 V=800.0 PL=0
MOVL C01702 V=800.0 PL=0
MOVL C01703 V=800.0 PL=0
MOVL C01704 V=800.0 PL=0
MOVL C01705 V=800.0 PL=0
MOVL C01706 V=800.0 PL=0
MOVL C01707 V=800.0 PL=0
MOVL C01708 V=800.0 PL=0
MOVL C01709 V=800.0 PL=0
MOVL C01710 V=800.0 PL=0
MOVL C01711 V=800.0 PL=0
MOVL C01712 V=800.0 PL=0
MOVL C01713 V=800.0 PL=0
MOVL C01714 V=800.0 PL=0
MOVL C01715 V=800.0 PL=0
MOVL C01716 V=800.0 PL=0
MOVL C01717 V=800.0 PL=0
MOVL C01718 V=800.0 PL=0
MOVL C01719 V=800.0 PL=0
MOVL C01720 V=800.0 PL=0
MOVL C01721 V=800.0 PL=0
MOVL C01722 V=800.0 PL=0
MOVL C01723 V=800.0 PL=0
MOVL C01724 V=800.0 PL=0
MOVL C01725 V=800.0 PL=0
MOVL C01726 V=800.0 PL=0
MOVL C01727 V=800.0 PL=0
MOVL C01728 V=800.0 PL=0
MOVL C01729 V=800.0 PL=0
MOVL C01730 V=800.0 PL=0
MOVL C01731 V=800.0 PL=0
MOVL C01732 V=800.0 PL=0
MOVL C01733 V=800.0 PL=0
MOVL C01734 V=800.0 PL=0
MOVL C01735 V=800.0 PL=0
MOVL C01736 V=800.0 PL=0
MOVL C01737 V=800.0 PL=0
MOVL C01738 V=800.0 PL=0
MOVL C01739 V=800.0 PL=0
MOVL C01740 V=800.0 PL=0
MOVL C01741 V=800.0 PL=0
MOVL C01742 V=800.0 PL=0
MOVL C01743 V=800.0 PL=0
MOVL C01744 V=800.0 PL=0
MOVL C01745 V=800.0 PL=0
MOVL C01746 V=800.0 PL=0
MOVL C01747 V=800.0 PL=0
MOVL C01748 V=800.0 PL=0
MOVL C01749 V=800.0 PL=0
MOVL C01750 V=800.0 PL=0
MOVL C01751 V=800.0 PL=0
MOVL C01752 V=800.0 PL=0
MOVL C01753 V=800.0 PL=0
MOVL C01754 V=800.0 PL=0
MOVL C01755 V=800.0 PL=0
MOVL C01756 V=800.0 PL=0
MOVL C01757 V=800.0 PL=0
MOVL C01758 V=800.0 PL=0
MOVL C01759 V=800.0 PL=0
MOVL C01760 V=800.0 PL=0
MOVL C01761 V=800.0 PL=0
MOVL C01762 V=800.0 PL=0
MOVL C01763 V=800.0 PL=0
MOVL C01764 V=800.0 PL=0
MOVL C01765 V=800.0 PL=0
MOVL C01766 V=800.0 PL=0
MOVL C01767 V=800.0 PL=0
MOVL C01768 V=800.0 PL=0
MOVL C01769 V=800.0 PL=0
MOVL C01770 V=800.0 PL=0
MOVL C01771 V=800.0 PL=0
MOVL C01772 V=800.0 PL=0
MOVL C01773 V=800.0 PL=0
MOVL C01774 V=800.0 PL=0
MOVL C01775 V=800.0 PL=0
MOVL C01776 V=800.0 PL=0
MOVL C01777 V=800.0 PL=0
MOVL C01778 V=800.0 PL=0
MOVL C01779 V=800.0 PL=0
MOVL C01780 V=800.0 PL=0
MOVL C01781 V=800.0 PL=0
MOVL C01782 V=800.0 PL=0
MOVL C01783 V=800.0 PL=0
MOVL C01784 V=800.0 PL=0
MOVL C01785 V=800.0 PL=0
MOVL C01786 V=800.0 PL=0
MOVL C01787 V=800.0 PL=0
MOVL C01788 V=800.0 PL=0
MOVL C01789 V=800.0 PL=0
MOVL C01790 V=800.0 PL=0
MOVL C01791 V=800.0 PL=0
MOVL C01792 V=800.0 PL=0
MOVL C01793 V=800.0 PL=0
MOVL C01794 V=800.0 PL=0
MOVL C01795 V=800.0 PL=0
MOVL C01796 V=800.0 PL=0
MOVL C01797 V=800.0 PL=0
MOVL C01798 V=800.0 PL=0
MOVL C01799 V=800.0 PL=0
MOVL C01800 V=800.0 PL=0
MOVL C01801 V=800.0 PL=0
MOVL C01802 V=800.0 PL=0
MOVL C01803 V=800.0 PL=0
MOVL C01804 V=800.0 PL=0
MOVL C01805 V=800.0 PL=0
MOVL C01806 V=800.0 PL=0
MOVL C01807 V=800.0 PL=0
MOVL C01808 V=800.0 PL=0
MOVL C01809 V=800.0 PL=0
MOVL C01810 V=800.0 PL=0
MOVL C01811 V=800.0 PL=0
MOVL C01812 V=800.0 PL=0
MOVL C01813 V=800.0 PL=0
MOVL C01814 V=800.0 PL=0
MOVL C01815 V=800.0 PL=0
MOVL C01816 V=800.0 PL=0
MOVL C01817 V=800.0 PL=0
MOVL C01818 V=800.0 PL=0
MOVL C01819 V=800.0 PL=0
MOVL C01820 V=800.0 PL=0
MOVL C01821 V=800.0 PL=0
MOVL C01822 V=800.0 PL=0
MOVL C01823 V=800.0 PL=0
MOVL C01824 V=800.0 PL=0
MOVL C01825 V=800.0 PL=0
MOVL C01826 V=800.0 PL=0
MOVL C01827 V=800.0 PL=0
MOVL C01828 V=800.0 PL=0
MOVL C01829 V=800.0 PL=0
MOVL C01830 V=800.0 PL=0
MOVL C01831 V=800.0 PL=0
MOVL C01832 V=800.0 PL=0
MOVL C01833 V=800.0 PL=0
MOVL C01834 V=800.0 PL=0
MOVL C01835 V=800.0 PL=0
MOVL C01836 V=800.0 PL=0
MOVL C01837 V=800.0 PL=0
MOVL C01838 V=800.0 PL=0
MOVL C01839 V=800.0 PL=0
MOVL C01840 V=800.0 PL=0
MOVL C01841 V=800.0 PL=0
MOVL C01842 V=800.0 PL=0
MOVL C01843 V=800.0 PL=0
MOVL C01844 V=800.0 PL=0
MOVL C01845 V=800.0 PL=0
MOVL C01846 V=800.0 PL=0
MOVL C01847 V=800.0 PL=0
MOVL C01848 V=800.0 PL=0
MOVL C01849 V=800.0 PL=0
MOVL C01850 V=800.0 PL=0
MOVL C01851 V=800.0 PL=0
MOVL C01852 V=800.0 PL=0
MOVL C01853 V=800.0 PL=0
MOVL C01854 V=800.0 PL=0
MOVL C01855 V=800.0 PL=0
MOVL C01856 V=800.0 PL=0
MOVL C01857 V=800.0 PL=0
MOVL C01858 V=800.0 PL=0
MOVL C01859 V=800.0 PL=0
MOVL C01860 V=800.0 PL=0
MOVL C01861 V=800.0 PL=0
MOVL C01862 V=800.0 PL=0
MOVL C01863 V=800.0 PL=0
MOVL C01864 V=800.0 PL=0
MOVL C01865 V=800.0 PL=0
MOVL C01866 V=800.0 PL=0
MOVL C01867 V=800.0 PL=0
MOVL C01868 V=800.0 PL=0
MOVL C01869 V=800.0 PL=0
MOVL C01870 V=800.0 PL=0
MOVL C01871 V=800.0 PL=0
MOVL C01872 V=800.0 PL=0
MOVL C01873 V=800.0 PL=0
MOVL C01874 V=800.0 PL=0
MOVL C01875 V=800.0 PL=0
MOVL C01876 V=800.0 PL=0
MOVL C01877 V=800.0 PL=0
MOVL C01878 V=800.0 PL=0
MOVL C01879 V=800.0 PL=0
MOVL C01880 V=800.0 PL=0
MOVL C01881 V=800.0 PL=0
MOVL C01882 V=800.0 PL=0
MOVL C01883 V=800.0 PL=0
MOVL C01884 V=800.0 PL=0
MOVL C01885 V=800.0 PL=0
MOVL C01886 V=800.0 PL=0
MOVL C01887 V=800.0 PL=0
MOVL C01888 V=800.0 PL=0
MOVL C01889 V=800.0 PL=0
MOVL C01890 V=800.0 PL=0
MOVL C01891 V=800.0 PL=0
MOVL C01892 V=800.0 PL=0
MOVL C01893 V=800.0 PL=0
MOVL C01894 V=800.0 PL=0
MOVL C01895 V=800.0 PL=0
MOVL C01896 V=800.0 PL=0
MOVL C01897 V=800.0 PL=0
MOVL C01898 V=800.0 PL=0
MOVL C01899 V=800.0 PL=0
MOVL C01900 V=800.0 PL=0
MOVL C01901 V=800.0 PL=0
MOVL C01902 V=800.0 PL=0
MOVL C01903 V=800.0 PL=0
MOVL C01904 V=800.0 PL=0
MOVL C01905 V=800.0 PL=0
